C01810=1071.589,307.374,406.167,174.565,30.421,155.473
C01811=1071.583,307.126,406.199,174.562,30.417,155.473
C01812=1071.577,306.878,406.231,174.558,30.412,155.472
C01813=1071.571,306.630,406.263,174.556,30.408,155.471
C01814=1071.564,306.382,406.295,174.552,30.403,155.470
C01815=1071.559,306.135,406.327,174.550,30.399,155.470
C01816=1071.553,305.887,406.359,174.547,30.395,155.469
C01817=1071.547,305.638,406.391,174.543,30.390,155.468
C01818=1071.540,305.390,406.422,174.541,30.386,155.467
C01819=1071.535,305.143,406.454,174.538,30.382,155.467
C01820=1071.529,304.895,406.487,174.535,30.377,155.466
C01821=1071.523,304.647,406.519,174.532,30.373,155.465
C01822=1071.516,304.400,406.550,174.529,30.368,155.464
C01823=1071.510,304.152,406.582,174.526,30.364,155.463
C01824=1071.503,303.847,406.621,174.522,30.359,155.463
C01825=1071.496,303.543,406.660,174.519,30.354,155.462
C01826=1071.488,303.240,406.699,174.515,30.348,155.461
C01827=1071.481,302.936,406.737,174.512,30.343,155.460
C01828=1071.475,302.687,406.769,174.508,30.338,155.459
C01829=1071.469,302.439,406.801,174.506,30.334,155.458
C01830=1071.463,302.192,406.833,174.503,30.330,155.457
C01831=1071.457,301.944,406.865,174.499,30.325,155.457
C01832=1071.452,301.696,406.896,174.497,30.321,155.456
C01833=1071.445,301.448,406.928,174.494,30.317,155.455
C01834=1071.440,301.201,406.959,174.492,30.313,155.454
C01835=1071.434,300.952,406.991,174.488,30.308,155.454
C01836=1071.427,300.704,407.022,174.485,30.304,155.453
C01837=1071.422,300.457,407.054,174.483,30.299,155.452
C01838=1071.416,300.208,407.086,174.479,30.295,155.451
C01839=1071.410,299.961,407.117,174.477,30.291,155.451
C01840=1071.404,299.713,407.149,174.474,30.287,155.450
C01841=1071.399,299.465,407.180,174.470,30.282,155.449
C01842=1071.392,299.217,407.211,174.468,30.278,155.448
C01843=1071.387,298.969,407.243,174.465,30.273,155.448
C01844=1071.380,298.721,407.274,174.463,30.270,155.447
C01845=1071.375,298.473,407.305,174.459,30.265,155.446
C01846=1071.369,298.225,407.337,174.456,30.261,155.445
C01847=1071.363,297.978,407.368,174.454,30.256,155.445
C01848=1071.357,297.729,407.400,174.450,30.252,155.444
C01849=1071.352,297.482,407.431,174.448,30.248,155.443
C01850=1071.345,297.234,407.463,174.445,30.243,155.442
C01851=1071.339,296.986,407.493,174.442,30.239,155.442
C01852=1071.333,296.738,407.525,174.439,30.235,155.441
C01853=1071.327,296.490,407.556,174.436,30.231,155.440
C01854=1071.321,296.242,407.588,174.434,30.226,155.439
C01855=1071.316,295.994,407.618,174.431,30.222,155.439
C01856=1071.309,295.746,407.649,174.427,30.218,155.438
C01857=1071.304,295.498,407.681,174.425,30.214,155.437
C01858=1071.297,295.250,407.712,174.422,30.210,155.436
C01859=1071.291,295.002,407.742,174.420,30.205,155.436
C01860=1071.285,294.754,407.773,174.416,30.201,155.435
C01861=1071.279,294.506,407.804,174.414,30.197,155.434
C01862=1071.273,294.259,407.835,174.411,30.193,155.434
C01863=1071.267,294.010,407.866,174.408,30.189,155.433
C01864=1071.262,293.763,407.898,174.405,30.184,155.432
C01865=1071.255,293.514,407.929,174.402,30.180,155.431
C01866=1071.249,293.266,407.959,174.400,30.176,155.431
C01867=1071.243,293.019,407.990,174.397,30.172,155.430
C01868=1071.237,292.771,408.021,174.393,30.167,155.429
C01869=1071.231,292.522,408.052,174.391,30.164,155.429
C01870=1071.225,292.275,408.083,174.388,30.159,155.428
C01871=1071.219,292.027,408.113,174.386,30.155,155.427
C01872=1071.213,291.778,408.144,174.382,30.151,155.426
C01873=1071.208,291.530,408.175,174.379,30.147,155.426
C01874=1071.202,291.283,408.206,174.377,30.143,155.425
C01875=1071.195,291.034,408.237,174.374,30.139,155.424
C01876=1071.190,290.820,408.264,174.372,30.135,155.424
C01877=1071.185,290.605,408.291,174.369,30.131,155.423
C01878=1071.180,290.390,408.316,174.366,30.128,155.422
C01879=1071.174,290.175,408.343,174.365,30.124,155.422
C01880=1071.169,289.960,408.370,174.362,30.120,155.421
C01881=1071.164,289.745,408.397,174.359,30.117,155.420
C01882=1071.159,289.530,408.423,174.357,30.113,155.420
C01883=1071.154,289.315,408.449,174.355,30.109,155.419
C01884=1071.148,289.068,408.480,174.352,30.105,155.419
C01885=1071.142,288.819,408.511,174.349,30.101,155.418
C01886=1071.136,288.571,408.541,174.346,30.097,155.417
C01887=1071.129,288.323,408.572,174.344,30.093,155.416
C01888=1071.124,288.076,408.603,174.341,30.089,155.416
C01889=1071.118,287.828,408.633,174.338,30.085,155.415
C01890=1071.111,287.579,408.664,174.335,30.080,155.414
C01891=1071.106,287.331,408.694,174.332,30.077,155.414
C01892=1071.099,287.084,408.724,174.330,30.073,155.413
C01893=1071.093,286.835,408.755,174.327,30.068,155.412
C01894=1071.087,286.587,408.784,174.324,30.064,155.411
C01895=1071.081,286.339,408.815,174.321,30.060,155.411
C01896=1071.075,286.091,408.845,174.318,30.056,155.410
C01897=1071.069,285.843,408.876,174.316,30.052,155.409
C01898=1071.063,285.595,408.906,174.313,30.048,155.409
C01899=1071.057,285.347,408.936,174.311,30.044,155.408
C01900=1071.052,285.099,408.967,174.307,30.040,155.407
C01901=1071.045,284.851,408.997,174.305,30.035,155.407
C01902=1071.039,284.603,409.028,174.302,30.032,155.406
C01903=1071.034,284.354,409.057,174.299,30.027,155.405
C01904=1071.028,284.107,409.088,174.297,30.023,155.404
C01905=1071.022,283.858,409.118,174.294,30.019,155.404
C01906=1071.015,283.611,409.148,174.291,30.015,155.403
C01907=1071.009,283.363,409.179,174.288,30.011,155.402
C01908=1071.004,283.114,409.208,174.286,30.007,155.402
C01909=1070.998,282.867,409.239,174.283,30.003,155.401
C01910=1070.991,282.618,409.269,174.280,29.999,155.400
C01911=1070.986,282.370,409.299,174.278,29.994,155.399
C01912=1070.980,282.122,409.329,174.275,29.991,155.399
C01913=1070.974,281.874,409.360,174.272,29.986,155.398
C01914=1070.969,281.625,409.389,174.269,29.982,155.397
C01915=1070.962,281.378,409.419,174.266,29.978,155.397
C01916=1070.956,281.129,409.450,174.264,29.974,155.396
C01917=1070.950,280.881,409.479,174.261,29.970,155.395
C01918=1070.945,280.633,409.510,174.259,29.966,155.395
C01919=1070.939,280.385,409.540,174.256,29.962,155.394
C01920=1070.932,280.137,409.569,174.254,29.958,155.393
C01921=1070.927,279.889,409.599,174.251,29.954,155.393
C01922=1070.921,279.641,409.629,174.248,29.949,155.392
C01923=1070.914,279.393,409.659,174.245,29.945,155.391
C01924=1070.908,279.144,409.689,174.242,29.942,155.391
C01925=1070.903,278.896,409.719,174.240,29.937,155.390
C01926=1070.896,278.648,409.748,174.237,29.933,155.389
C01927=1070.891,278.401,409.779,174.235,29.929,155.388
C01928=1070.885,278.152,409.808,174.232,29.926,155.388
C01929=1070.879,277.904,409.837,174.229,29.921,155.387
C01930=1070.873,277.656,409.868,174.227,29.917,155.386
C01931=1070.867,277.408,409.897,174.223,29.913,155.386
C01932=1070.857,276.988,409.948,174.219,29.906,155.384
C01933=1070.846,276.569,409.998,174.215,29.899,155.383
C01934=1070.836,276.149,410.048,174.210,29.893,155.382
C01935=1070.826,275.729,410.098,174.206,29.886,155.381
C01936=1070.821,275.481,410.128,174.204,29.882,155.380
C01937=1070.814,275.233,410.157,174.200,29.878,155.380
C01938=1070.809,274.985,410.187,174.198,29.873,155.379
C01939=1070.803,274.737,410.216,174.195,29.869,155.378
C01940=1070.797,274.489,410.246,174.192,29.866,155.378
C01941=1070.790,274.241,410.275,174.190,29.862,155.377
C01942=1070.785,273.992,410.305,174.187,29.857,155.376
C01943=1070.779,273.744,410.334,174.185,29.853,155.376
C01944=1070.773,273.496,410.364,174.182,29.849,155.375
C01945=1070.768,273.247,410.393,174.180,29.846,155.374
C01946=1070.761,273.000,410.423,174.177,29.841,155.373
C01947=1070.755,272.752,410.452,174.174,29.837,155.373
C01948=1070.749,272.503,410.482,174.172,29.833,155.372
C01949=1070.743,272.255,410.511,174.169,29.829,155.371
C01950=1070.738,272.007,410.541,174.167,29.826,155.371
C01951=1070.731,271.758,410.570,174.164,29.821,155.370
C01952=1070.725,271.510,410.599,174.162,29.817,155.369
C01953=1070.720,271.262,410.628,174.159,29.813,155.369
C01954=1070.713,271.014,410.657,174.156,29.809,155.368
C01955=1070.708,270.765,410.687,174.153,29.805,155.367
C01956=1070.702,270.517,410.716,174.150,29.801,155.367
C01957=1070.696,270.270,410.745,174.148,29.797,155.366
C01958=1070.690,270.021,410.774,174.145,29.793,155.365
C01959=1070.684,269.773,410.803,174.143,29.789,155.365
C01960=1070.678,269.525,410.832,174.140,29.785,155.364
C01961=1070.672,269.277,410.862,174.138,29.781,155.363
C01962=1070.666,269.028,410.891,174.135,29.777,155.363
C01963=1070.660,268.780,410.920,174.132,29.773,155.362
C01964=1070.654,268.532,410.950,174.130,29.769,155.361
C01965=1070.648,268.284,410.979,174.127,29.765,155.361
C01966=1070.642,268.035,411.007,174.125,29.761,155.360
C01967=1070.636,267.787,411.036,174.122,29.757,155.359
C01968=1070.630,267.539,411.065,174.120,29.753,155.359
C01969=1070.625,267.291,411.094,174.117,29.749,155.358
C01970=1070.619,267.043,411.123,174.115,29.745,155.357
C01971=1070.613,266.794,411.152,174.112,29.741,155.357
C01972=1070.606,266.546,411.181,174.109,29.738,155.356
C01973=1070.601,266.297,411.210,174.107,29.733,155.355
C01974=1070.595,266.049,411.239,174.104,29.729,155.355
C01975=1070.589,265.801,411.268,174.102,29.725,155.354
C01976=1070.583,265.553,411.296,174.099,29.721,155.353
C01977=1070.577,265.305,411.326,174.097,29.717,155.353
C01978=1070.571,265.057,411.355,174.094,29.713,155.352
C01979=1070.565,264.808,411.383,174.092,29.709,155.351
C01980=1070.559,264.560,411.413,174.089,29.705,155.351
C01981=1070.553,264.312,411.442,174.087,29.701,155.350
C01982=1070.547,264.064,411.470,174.084,29.697,155.349
C01983=1070.541,263.815,411.499,174.081,29.694,155.349
C01984=1070.531,263.399,411.547,174.077,29.686,155.347
C01985=1070.521,262.982,411.594,174.073,29.680,155.346
C01986=1070.511,262.566,411.643,174.069,29.673,155.345
C01987=1070.501,262.150,411.691,174.064,29.667,155.344
C01988=1070.495,261.901,411.719,174.062,29.663,155.343
C01989=1070.489,261.654,411.748,174.059,29.659,155.343
C01990=1070.483,261.405,411.776,174.057,29.655,155.342
C01991=1070.477,261.157,411.805,174.054,29.651,155.342
C01992=1070.470,260.909,411.833,174.052,29.647,155.341
C01993=1070.464,260.661,411.862,174.049,29.643,155.340
C01994=1070.458,260.412,411.890,174.047,29.640,155.340
C01995=1070.453,260.164,411.918,174.044,29.636,155.339
C01996=1070.446,259.916,411.947,174.042,29.632,155.338
C01997=1070.440,259.667,411.975,174.040,29.628,155.338
C01998=1070.434,259.419,412.004,174.037,29.624,155.337
C01999=1070.428,259.171,412.032,174.035,29.620,155.336
C02000=1070.422,258.922,412.060,174.032,29.616,155.336
C02001=1070.416,258.674,412.089,174.030,29.612,155.335
C02002=1070.410,258.425,412.117,174.027,29.608,155.334
C02003=1070.405,258.177,412.145,174.025,29.604,155.334
C02004=1070.399,257.929,412.174,174.022,29.601,155.333
C02005=1070.392,257.681,412.202,174.019,29.597,155.332
C02006=1070.386,257.433,412.230,174.017,29.592,155.332
C02007=1070.380,257.184,412.259,174.014,29.588,155.331
C02008=1070.374,256.935,412.287,174.012,29.584,155.330
C02009=1070.369,256.688,412.316,174.009,29.580,155.330
C02010=1070.362,256.439,412.343,174.007,29.576,155.329
C02011=1070.356,256.191,412.372,174.004,29.573,155.328
C02012=1070.351,255.943,412.400,174.003,29.569,155.328
C02013=1070.345,255.694,412.428,174.000,29.565,155.327
C02014=1070.339,255.445,412.456,173.998,29.561,155.326
C02015=1070.333,255.198,412.484,173.995,29.557,155.326
C02016=1070.327,254.949,412.513,173.993,29.553,155.325
C02017=1070.321,254.700,412.541,173.990,29.549,155.325
C02018=1070.315,254.452,412.569,173.988,29.545,155.324
C02019=1070.309,254.204,412.597,173.985,29.541,155.323
C02020=1070.303,253.956,412.625,173.982,29.537,155.322
C02021=1070.297,253.707,412.653,173.980,29.533,155.322
C02022=1070.291,253.458,412.681,173.978,29.529,155.321
C02023=1070.285,253.211,412.709,173.976,29.525,155.320
C02024=1070.279,252.962,412.737,173.973,29.521,155.320
C02025=1070.274,252.714,412.765,173.971,29.517,155.319
C02026=1070.268,252.465,412.793,173.968,29.513,155.318
C02027=1070.261,252.217,412.821,173.966,29.509,155.318
C02028=1070.256,251.969,412.849,173.963,29.505,155.317
C02029=1070.250,251.720,412.877,173.961,29.501,155.316
C02030=1070.245,251.472,412.905,173.958,29.497,155.316
C02031=1070.238,251.223,412.933,173.957,29.494,155.315
C02032=1070.233,250.975,412.961,173.954,29.490,155.315
C02033=1070.227,250.726,412.989,173.952,29.485,155.314
C02034=1070.221,250.478,413.017,173.949,29.481,155.313
C02035=1070.215,250.229,413.044,173.947,29.477,155.312
C02036=1070.205,249.811,413.091,173.942,29.471,155.311
C02037=1070.196,249.392,413.138,173.938,29.464,155.310
C02038=1070.186,248.974,413.185,173.935,29.457,155.309
C02039=1070.176,248.555,413.232,173.931,29.451,155.308
C02040=1070.170,248.307,413.260,173.928,29.446,155.307
C02041=1070.165,248.059,413.288,173.926,29.442,155.307
C02042=1070.159,247.810,413.315,173.923,29.438,155.306
C02043=1070.153,247.562,413.343,173.921,29.434,155.305
C02044=1070.147,247.313,413.371,173.919,29.431,155.305
C02045=1070.142,247.065,413.398,173.917,29.426,155.304
C02046=1070.135,246.816,413.426,173.914,29.422,155.303
C02047=1070.130,246.568,413.454,173.912,29.418,155.303
C02048=1070.124,246.320,413.481,173.909,29.414,155.302
C02049=1070.118,246.071,413.509,173.907,29.410,155.301
C02050=1070.112,245.823,413.536,173.905,29.407,155.301
C02051=1070.107,245.574,413.564,173.902,29.403,155.300
C02052=1070.101,245.326,413.591,173.900,29.399,155.299
C02053=1070.094,245.078,413.619,173.897,29.395,155.299
C02054=1070.089,244.829,413.646,173.895,29.390,155.298
C02055=1070.083,244.581,413.674,173.892,29.386,155.297
C02056=1070.077,244.332,413.701,173.891,29.383,155.297
C02057=1070.071,244.084,413.729,173.888,29.379,155.296
C02058=1070.065,243.835,413.756,173.886,29.375,155.295
C02059=1070.059,243.587,413.784,173.883,29.371,155.295
C02060=1070.054,243.339,413.811,173.881,29.367,155.294
C02061=1070.048,243.090,413.839,173.879,29.363,155.293
C02062=1070.042,242.842,413.865,173.877,29.359,155.293
C02063=1070.037,242.594,413.893,173.874,29.355,155.292
C02064=1070.030,242.345,413.920,173.872,29.351,155.291
C02065=1070.024,242.097,413.948,173.869,29.347,155.291
C02066=1070.018,241.847,413.975,173.868,29.343,155.290
C02067=1070.013,241.599,414.002,173.865,29.339,155.289
C02068=1070.006,241.351,414.030,173.863,29.335,155.289
C02069=1070.000,241.102,414.056,173.860,29.331,155.288
C02070=1069.994,240.854,414.083,173.858,29.327,155.287
C02071=1069.989,240.605,414.111,173.856,29.324,155.287
C02072=1069.983,240.357,414.138,173.854,29.320,155.286
C02073=1069.977,240.108,414.164,173.851,29.316,155.285
C02074=1069.970,239.860,414.192,173.849,29.312,155.285
C02075=1069.965,239.611,414.219,173.846,29.308,155.284
C02076=1069.959,239.363,414.246,173.845,29.304,155.284
C02077=1069.953,239.115,414.274,173.842,29.300,155.283
C02078=1069.947,238.866,414.300,173.840,29.296,155.282
C02079=1069.941,238.618,414.327,173.837,29.292,155.281
C02080=1069.935,238.369,414.354,173.835,29.288,155.281
C02081=1069.930,238.120,414.381,173.833,29.284,155.280
C02082=1069.924,237.872,414.409,173.831,29.280,155.280
C02083=1069.917,237.623,414.436,173.828,29.276,155.279
C02084=1069.912,237.375,414.462,173.826,29.272,155.278
C02085=1069.906,237.127,414.489,173.824,29.268,155.278
C02086=1069.900,236.878,414.516,173.822,29.264,155.277
C02087=1069.894,236.629,414.543,173.819,29.260,155.276
C02088=1069.889,236.417,414.566,173.818,29.257,155.276
C02089=1069.884,236.205,414.589,173.815,29.253,155.275
C02090=1069.879,235.992,414.612,173.813,29.250,155.275
C02091=1069.875,235.780,414.635,173.812,29.247,155.274
C02092=1069.869,235.567,414.658,173.809,29.243,155.273
C02093=1069.864,235.354,414.681,173.808,29.240,155.273
C02094=1069.859,235.142,414.704,173.806,29.236,155.272
C02095=1069.854,234.929,414.727,173.804,29.233,155.272
C02096=1069.848,234.681,414.754,173.801,29.229,155.271
C02097=1069.842,234.432,414.781,173.800,29.225,155.270
C02098=1069.836,234.184,414.808,173.797,29.221,155.270
C02099=1069.830,233.936,414.834,173.795,29.217,155.269
C02100=1069.824,233.687,414.861,173.792,29.213,155.268
C02101=1069.819,233.439,414.888,173.791,29.209,155.268
C02102=1069.813,233.189,414.914,173.788,29.205,155.267
C02103=1069.807,232.941,414.940,173.786,29.201,155.266
C02104=1069.801,232.693,414.967,173.783,29.197,155.266
C02105=1069.795,232.444,414.994,173.782,29.193,155.265
C02106=1069.790,232.196,415.020,173.779,29.189,155.265
C02107=1069.783,231.947,415.047,173.777,29.185,155.264
C02108=1069.777,231.698,415.074,173.775,29.181,155.263
C02109=1069.772,231.450,415.101,173.773,29.177,155.262
C02110=1069.766,231.202,415.127,173.770,29.173,155.262
C02111=1069.760,230.953,415.154,173.768,29.169,155.261
C02112=1069.755,230.704,415.180,173.766,29.166,155.260
C02113=1069.749,230.456,415.207,173.764,29.162,155.260
C02114=1069.743,230.208,415.233,173.761,29.158,155.259
C02115=1069.737,229.959,415.260,173.760,29.154,155.259
C02116=1069.730,229.711,415.286,173.757,29.149,155.258
C02117=1069.725,229.462,415.312,173.755,29.145,155.257
C02118=1069.719,229.213,415.339,173.752,29.141,155.257
C02119=1069.713,228.965,415.366,173.751,29.138,155.256
C02120=1069.707,228.717,415.392,173.748,29.134,155.255
C02121=1069.701,228.467,415.418,173.746,29.130,155.255
C02122=1069.695,228.219,415.445,173.744,29.126,155.254
C02123=1069.689,227.970,415.471,173.742,29.122,155.253
C02124=1069.683,227.722,415.497,173.739,29.118,155.253
C02125=1069.677,227.473,415.523,173.737,29.114,155.252
C02126=1069.671,227.225,415.550,173.735,29.110,155.251
C02127=1069.666,226.976,415.576,173.733,29.106,155.251
C02128=1069.659,226.728,415.602,173.730,29.102,155.250
C02129=1069.654,226.480,415.628,173.729,29.098,155.249
C02130=1069.647,226.230,415.655,173.726,29.094,155.249
C02131=1069.642,225.982,415.681,173.724,29.090,155.248
C02132=1069.635,225.733,415.707,173.722,29.086,155.247
C02133=1069.630,225.485,415.733,173.720,29.082,155.247
C02134=1069.624,225.236,415.759,173.718,29.078,155.246
C02135=1069.618,224.988,415.785,173.716,29.074,155.245
C02136=1069.612,224.739,415.811,173.714,29.070,155.245
C02137=1069.606,224.490,415.838,173.711,29.066,155.244
C02138=1069.600,224.242,415.864,173.710,29.062,155.243
C02139=1069.595,223.993,415.890,173.707,29.058,155.243
C02140=1069.589,223.744,415.916,173.705,29.054,155.242
C02141=1069.583,223.496,415.942,173.703,29.050,155.241
C02142=1069.577,223.247,415.968,173.701,29.046,155.241
C02143=1069.571,222.999,415.995,173.698,29.042,155.240
C02144=1069.566,222.783,416.017,173.697,29.039,155.239
C02145=1069.561,222.566,416.040,173.695,29.035,155.239
C02146=1069.556,222.350,416.062,173.693,29.031,155.238
C02147=1069.551,222.132,416.085,173.691,29.028,155.238
C02148=1069.546,221.916,416.107,173.690,29.025,155.237
C02149=1069.541,221.699,416.131,173.687,29.021,155.237
C02150=1069.536,221.483,416.153,173.686,29.018,155.236
C02151=1069.531,221.266,416.176,173.684,29.015,155.235
C02152=1069.525,221.017,416.201,173.682,29.010,155.235
C02153=1069.519,220.768,416.227,173.679,29.006,155.234
C02154=1069.513,220.520,416.253,173.678,29.002,155.233
C02155=1069.507,220.271,416.279,173.675,28.998,155.233
C02156=1069.501,220.023,416.304,173.673,28.994,155.232
C02157=1069.494,219.775,416.331,173.671,28.991,155.231
C02158=1069.489,219.526,416.356,173.669,28.987,155.231
C02159=1069.483,219.277,416.382,173.667,28.983,155.230
C02160=1069.477,219.028,416.408,173.665,28.979,155.230
C02161=1069.471,218.780,416.434,173.662,28.975,155.229
C02162=1069.465,218.531,416.460,173.661,28.970,155.228
C02163=1069.459,218.282,416.485,173.658,28.966,155.227
C02164=1069.453,218.034,416.510,173.656,28.962,155.227
C02165=1069.448,217.785,416.536,173.654,28.959,155.226
C02166=1069.441,217.537,416.562,173.652,28.955,155.226
C02167=1069.436,217.288,416.588,173.650,28.951,155.225
C02168=1069.430,217.040,416.613,173.648,28.947,155.224
C02169=1069.424,216.791,416.639,173.646,28.942,155.223
C02170=1069.418,216.542,416.665,173.644,28.939,155.223
C02171=1069.412,216.293,416.690,173.642,28.935,155.222
C02172=1069.406,216.044,416.716,173.639,28.931,155.222
C02173=1069.401,215.796,416.741,173.638,28.927,155.221
C02174=1069.395,215.548,416.766,173.635,28.922,155.220
C02175=1069.389,215.299,416.793,173.634,28.919,155.219
C02176=1069.383,215.051,416.818,173.631,28.914,155.219
C02177=1069.377,214.802,416.844,173.629,28.910,155.218
C02178=1069.371,214.553,416.869,173.627,28.907,155.218
C02179=1069.365,214.305,416.894,173.625,28.902,155.217
C02180=1069.360,214.056,416.920,173.624,28.898,155.216
C02181=1069.354,213.808,416.946,173.621,28.894,155.215
C02182=1069.348,213.559,416.971,173.619,28.890,155.215
C02183=1069.342,213.310,416.997,173.617,28.886,155.214
C02184=1069.336,213.062,417.022,173.615,28.882,155.213
C02185=1069.330,212.813,417.047,173.613,28.878,155.213
C02186=1069.325,212.564,417.073,173.611,28.874,155.212
C02187=1069.319,212.315,417.098,173.608,28.870,155.211
C02188=1069.313,212.066,417.123,173.607,28.866,155.211
C02189=1069.306,211.818,417.148,173.605,28.862,155.210
C02190=1069.301,211.570,417.173,173.603,28.858,155.209
C02191=1069.295,211.321,417.199,173.601,28.854,155.209
C02192=1069.289,211.072,417.225,173.599,28.850,155.208
C02193=1069.283,210.823,417.250,173.597,28.846,155.207
C02194=1069.277,210.575,417.275,173.594,28.842,155.207
C02195=1069.271,210.326,417.300,173.593,28.838,155.206
C02196=1069.265,210.077,417.325,173.590,28.834,155.205
C02197=1069.260,209.828,417.351,173.589,28.830,155.205
C02198=1069.254,209.580,417.376,173.587,28.826,155.204
C02199=1069.248,209.332,417.401,173.585,28.822,155.203
C02200=1069.243,209.117,417.423,173.583,28.818,155.203
C02201=1069.237,208.903,417.444,173.581,28.815,155.202
C02202=1069.232,208.688,417.466,173.580,28.811,155.202
C02203=1069.228,208.474,417.487,173.578,28.808,155.201
C02204=1069.223,208.259,417.509,173.576,28.804,155.200
C02205=1069.218,208.046,417.531,173.574,28.801,155.200
C02206=1069.212,207.831,417.552,173.572,28.798,155.199
C02207=1069.207,207.616,417.574,173.571,28.794,155.199
C02208=1069.183,206.573,417.677,173.428,28.722,155.196
C02209=1069.177,206.324,417.701,173.427,28.718,155.195
C02210=1069.171,206.076,417.725,173.424,28.715,155.195
C02211=1069.166,205.827,417.749,173.422,28.712,155.194
C02212=1069.160,205.578,417.774,173.420,28.709,155.194
C02213=1069.155,205.329,417.798,173.418,28.706,155.193
C02214=1069.148,205.080,417.822,173.415,28.703,155.193
C02215=1069.143,204.832,417.846,173.414,28.700,155.192
C02216=1069.138,204.583,417.871,173.411,28.697,155.192
C02217=1069.132,204.334,417.895,173.409,28.693,155.191
C02218=1069.126,204.086,417.919,173.407,28.690,155.191
C02219=1069.120,203.837,417.943,173.404,28.687,155.190
C02220=1069.115,203.588,417.968,173.402,28.684,155.190
C02221=1069.109,203.339,417.992,173.400,28.681,155.190
C02222=1069.103,203.091,418.016,173.398,28.678,155.189
C02223=1069.097,202.842,418.040,173.395,28.675,155.189
C02224=1069.092,202.593,418.065,173.394,28.672,155.188
C02225=1069.087,202.344,418.089,173.391,28.669,155.188
C02226=1069.080,202.095,418.113,173.389,28.665,155.187
C02227=1069.075,201.847,418.137,173.387,28.662,155.187
C02228=1069.069,201.598,418.160,173.384,28.660,155.187
C02229=1069.063,201.349,418.185,173.382,28.656,155.186
C02230=1069.057,201.100,418.208,173.380,28.653,155.186
C02231=1069.052,200.852,418.233,173.378,28.650,155.185
C02232=1069.045,200.603,418.257,173.376,28.647,155.185
C02233=1069.040,200.354,418.281,173.374,28.644,155.184
C02234=1069.034,200.105,418.304,173.371,28.641,155.184
C02235=1069.028,199.856,418.328,173.370,28.638,155.183
C02236=1069.022,199.608,418.352,173.367,28.635,155.183
C02237=1069.017,199.359,418.376,173.364,28.632,155.183
C02238=1069.011,199.110,418.400,173.363,28.629,155.182
C02239=1069.005,198.861,418.423,173.360,28.626,155.182
C02240=1068.999,198.613,418.448,173.359,28.623,155.181
C02241=1068.993,198.364,418.472,173.356,28.620,155.181
C02242=1068.988,198.115,418.495,173.354,28.617,155.180
C02243=1068.982,197.866,418.519,173.352,28.614,155.180
C02244=1068.976,197.618,418.543,173.350,28.611,155.180
C02245=1068.970,197.368,418.566,173.348,28.608,155.179
C02246=1068.965,197.119,418.591,173.345,28.605,155.179
C02247=1068.959,196.871,418.614,173.343,28.602,155.178
C02248=1068.952,196.622,418.638,173.341,28.599,155.178
C02249=1068.947,196.373,418.662,173.339,28.596,155.177
C02250=1068.941,196.125,418.685,173.337,28.593,155.177
C02251=1068.936,195.876,418.709,173.335,28.590,155.177
C02252=1068.930,195.627,418.733,173.332,28.587,155.176
C02253=1068.924,195.378,418.757,173.331,28.584,155.176
C02254=1068.918,195.129,418.780,173.328,28.581,155.175
C02255=1068.912,194.881,418.804,173.326,28.578,155.175
C02256=1068.907,194.632,418.827,173.324,28.575,155.174
C02257=1068.901,194.383,418.851,173.322,28.572,155.174
C02258=1068.896,194.133,418.875,173.320,28.569,155.173
C02259=1068.890,193.885,418.899,173.317,28.566,155.173
C02260=1068.884,193.636,418.922,173.316,28.563,155.173
C02261=1068.879,193.388,418.946,173.313,28.560,155.172
C02262=1068.873,193.139,418.969,173.312,28.557,155.172
C02263=1068.868,192.890,418.993,173.309,28.554,155.171
C02264=1068.861,192.641,419.016,173.307,28.551,155.171
C02265=1068.855,192.392,419.040,173.305,28.548,155.170
C02266=1068.850,192.143,419.064,173.303,28.545,155.170
C02267=1068.844,191.895,419.087,173.301,28.542,155.170
C02268=1068.838,191.646,419.110,173.298,28.538,155.169
C02269=1068.832,191.363,419.138,173.297,28.536,155.169
C02270=1068.826,191.081,419.164,173.294,28.532,155.168
C02271=1068.819,190.799,419.191,173.292,28.529,155.168
C02272=1068.813,190.517,419.217,173.289,28.525,155.167
C02273=1068.808,190.268,419.241,173.287,28.522,155.167
C02274=1068.802,190.020,419.264,173.285,28.519,155.166
C02275=1068.796,189.771,419.287,173.283,28.516,155.166
C02276=1068.791,189.521,419.311,173.281,28.513,155.165
C02277=1068.785,189.273,419.334,173.279,28.510,155.165
C02278=1068.779,189.024,419.357,173.277,28.507,155.165
C02279=1068.774,188.775,419.381,173.274,28.504,155.164
C02280=1068.768,188.526,419.405,173.273,28.501,155.164
C02281=1068.762,188.277,419.428,173.270,28.498,155.163
C02282=1068.757,188.028,419.451,173.269,28.495,155.163
C02283=1068.751,187.779,419.474,173.266,28.492,155.162
C02284=1068.745,187.531,419.498,173.265,28.489,155.162
C02285=1068.739,187.282,419.521,173.262,28.486,155.161
C02286=1068.734,187.033,419.544,173.261,28.483,155.161
C02287=1068.729,186.784,419.567,173.258,28.480,155.161
C02288=1068.723,186.536,419.591,173.257,28.477,155.160
C02289=1068.718,186.286,419.615,173.254,28.474,155.160
C02290=1068.712,186.037,419.638,173.252,28.471,155.159
C02291=1068.706,185.789,419.661,173.250,28.468,155.159
C02292=1068.700,185.540,419.683,173.248,28.465,155.158
C02293=1068.695,185.291,419.708,173.246,28.462,155.158
C02294=1068.689,185.042,419.731,173.244,28.459,155.158
C02295=1068.684,184.793,419.754,173.242,28.456,155.157
C02296=1068.678,184.544,419.777,173.240,28.453,155.157
C02297=1068.672,184.295,419.800,173.238,28.450,155.156
C02298=1068.666,184.047,419.822,173.236,28.448,155.156
C02299=1068.661,183.798,419.845,173.233,28.445,155.156
C02300=1068.655,183.549,419.868,173.232,28.442,155.155
C02301=1068.649,183.300,419.891,173.229,28.439,155.155
C02302=1068.644,183.051,419.914,173.228,28.436,155.154
C02303=1068.637,182.802,419.937,173.225,28.433,155.154
C02304=1068.631,182.554,419.960,173.224,28.430,155.153
C02305=1068.626,182.305,419.982,173.221,28.427,155.153
C02306=1068.620,182.056,420.005,173.220,28.424,155.153
C02307=1068.614,181.807,420.028,173.218,28.422,155.152
C02308=1068.608,181.558,420.051,173.215,28.419,155.152
C02309=1068.602,181.309,420.074,173.214,28.416,155.151
C02310=1068.596,181.060,420.097,173.211,28.413,155.151
C02311=1068.591,180.812,420.120,173.210,28.410,155.151
C02312=1068.585,180.563,420.143,173.207,28.407,155.150
C02313=1068.579,180.314,420.165,173.206,28.405,155.150
C02314=1068.573,180.065,420.188,173.203,28.402,155.149
C02315=1068.567,179.816,420.211,173.201,28.399,155.149
C02316=1068.561,179.567,420.234,173.199,28.396,155.149
C02317=1068.556,179.318,420.256,173.197,28.393,155.148
C02318=1068.550,179.069,420.279,173.195,28.390,155.148
C02319=1068.544,178.820,420.302,173.193,28.387,155.147
C02320=1068.538,178.571,420.324,173.192,28.385,155.147
C02321=1068.532,178.323,420.347,173.189,28.382,155.147
C02322=1068.526,178.074,420.370,173.187,28.379,155.146
C02323=1068.521,177.825,420.393,173.185,28.376,155.146
C02324=1068.515,177.575,420.415,173.183,28.373,155.145
C02325=1068.509,177.327,420.438,173.181,28.370,155.145
C02326=1068.503,177.078,420.461,173.179,28.367,155.145
C02327=1068.497,176.829,420.483,173.178,28.364,155.144
C02328=1068.492,176.579,420.506,173.175,28.361,155.144
C02329=1068.485,176.331,420.528,173.174,28.359,155.143
C02330=1068.480,176.082,420.551,173.171,28.356,155.143
C02331=1068.474,175.834,420.574,173.169,28.353,155.143
C02332=1068.469,175.584,420.596,173.167,28.350,155.142
C02333=1068.462,175.301,420.621,173.165,28.347,155.142
C02334=1068.456,175.019,420.647,173.163,28.344,155.141
C02335=1068.449,174.736,420.673,173.160,28.340,155.141
C02336=1068.442,174.454,420.698,173.158,28.337,155.140
C02337=1068.437,174.205,420.721,173.156,28.334,155.140
C02338=1068.431,173.956,420.744,173.155,28.331,155.139
C02339=1068.425,173.707,420.766,173.152,28.328,155.139
C02340=1068.420,173.459,420.788,173.151,28.326,155.139
C02341=1068.414,173.210,420.811,173.148,28.323,155.138
C02342=1068.408,172.960,420.833,173.147,28.320,155.138
C02343=1068.402,172.712,420.856,173.145,28.317,155.137
C02344=1068.397,172.462,420.878,173.143,28.314,155.137
C02345=1068.391,172.213,420.901,173.141,28.311,155.137
C02346=1068.385,171.965,420.923,173.139,28.309,155.136
C02347=1068.380,171.716,420.945,173.137,28.306,155.136
C02348=1068.374,171.467,420.968,173.135,28.303,155.135
C02349=1068.368,171.217,420.990,173.133,28.299,155.135
C02350=1068.363,170.970,421.012,173.131,28.297,155.135
C02351=1068.357,170.720,421.034,173.130,28.294,155.134
C02352=1068.351,170.471,421.057,173.127,28.291,155.134
C02353=1068.345,170.222,421.079,173.126,28.288,155.133
C02354=1068.339,169.973,421.102,173.123,28.285,155.133
C02355=1068.335,169.724,421.124,173.121,28.283,155.133
C02356=1068.328,169.476,421.146,173.120,28.280,155.132
C02357=1068.323,169.226,421.168,173.117,28.277,155.132
C02358=1068.318,168.978,421.191,173.116,28.274,155.131
C02359=1068.311,168.729,421.213,173.114,28.271,155.131
C02360=1068.306,168.480,421.236,173.112,28.268,155.130
C02361=1068.300,168.230,421.258,173.110,28.265,155.130
C02362=1068.294,167.982,421.280,173.109,28.262,155.130
C02363=1068.289,167.733,421.302,173.106,28.259,155.129
C02364=1068.284,167.483,421.324,173.104,28.257,155.129
C02365=1068.278,167.235,421.346,173.103,28.254,155.128
C02366=1068.272,166.986,421.368,173.100,28.251,155.128
C02367=1068.267,166.737,421.391,173.099,28.248,155.128
C02368=1068.260,166.488,421.413,173.097,28.245,155.127
C02369=1068.256,166.239,421.435,173.095,28.242,155.127
C02370=1068.250,165.990,421.458,173.093,28.239,155.126
C02371=1068.244,165.742,421.479,173.092,28.236,155.126
C02372=1068.239,165.492,421.501,173.089,28.233,155.125
C02373=1068.233,165.243,421.524,173.088,28.231,155.125
C02374=1068.228,164.995,421.546,173.086,28.228,155.125
C02375=1068.222,164.745,421.568,173.083,28.225,155.124
C02376=1068.216,164.497,421.590,173.082,28.222,155.124
C02377=1068.211,164.248,421.612,173.080,28.219,155.123
C02378=1068.205,163.998,421.634,173.078,28.216,155.123
C02379=1068.199,163.749,421.656,173.076,28.213,155.123
C02380=1068.194,163.501,421.678,173.075,28.211,155.122
C02381=1068.188,163.252,421.700,173.072,28.208,155.122
C02382=1068.183,163.003,421.722,173.071,28.205,155.121
C02383=1068.178,162.753,421.744,173.069,28.202,155.121
C02384=1068.171,162.505,421.767,173.067,28.199,155.120
C02385=1068.166,162.256,421.788,173.065,28.196,155.120
C02386=1068.160,162.007,421.810,173.064,28.193,155.120
C02387=1068.155,161.758,421.832,173.061,28.190,155.119
C02388=1068.150,161.508,421.854,173.059,28.187,155.119
C02389=1068.144,161.260,421.875,173.058,28.185,155.118
C02390=1068.139,161.011,421.898,173.055,28.182,155.118
C02391=1068.133,160.762,421.920,173.054,28.179,155.118
C02392=1068.127,160.513,421.941,173.052,28.176,155.117
C02393=1068.121,160.264,421.963,173.051,28.173,155.117
C02394=1068.115,160.015,421.985,173.048,28.170,155.116
C02395=1068.110,159.766,422.006,173.047,28.168,155.116
C02396=1068.104,159.517,422.028,173.045,28.165,155.116
C02397=1068.097,159.234,422.052,173.043,28.161,155.115
C02398=1068.091,158.950,422.078,173.040,28.158,155.115
C02399=1068.085,158.668,422.102,173.039,28.155,155.114
C02400=1068.078,158.385,422.126,173.036,28.152,155.114
C02401=1068.072,158.136,422.148,173.035,28.149,155.113
C02402=1068.066,157.887,422.170,173.033,28.147,155.113
C02403=1068.061,157.638,422.192,173.030,28.144,155.113
C02404=1068.055,157.389,422.213,173.029,28.141,155.112
C02405=1068.049,157.140,422.234,173.027,28.138,155.112
C02406=1068.043,156.891,422.256,173.026,28.135,155.111
C02407=1068.038,156.642,422.278,173.023,28.132,155.111
C02408=1068.032,156.393,422.300,173.022,28.130,155.111
C02409=1068.026,156.144,422.321,173.020,28.127,155.110
C02410=1068.020,155.895,422.342,173.018,28.124,155.110
C02411=1068.015,155.646,422.365,173.016,28.121,155.109
C02412=1068.009,155.397,422.386,173.014,28.118,155.109
C02413=1068.003,155.148,422.408,173.013,28.116,155.109
C02414=1067.998,154.899,422.429,173.010,28.113,155.108
C02415=1067.992,154.650,422.450,173.009,28.110,155.108
C02416=1067.986,154.402,422.472,173.007,28.107,155.107
C02417=1067.980,154.152,422.493,173.006,28.104,155.107
C02418=1067.974,153.903,422.514,173.003,28.101,155.107
C02419=1067.969,153.654,422.536,173.002,28.099,155.106
C02420=1067.963,153.405,422.558,173.000,28.096,155.106
C02421=1067.957,153.156,422.579,172.998,28.093,155.105
C02422=1067.951,152.907,422.601,172.996,28.090,155.105
C02423=1067.946,152.658,422.621,172.994,28.087,155.105
C02424=1067.940,152.409,422.643,172.993,28.085,155.104
C02425=1067.934,152.160,422.664,172.990,28.082,155.104
C02426=1067.928,151.911,422.686,172.989,28.079,155.104
C02427=1067.923,151.662,422.706,172.987,28.077,155.103
C02428=1067.917,151.413,422.728,172.986,28.074,155.103
C02429=1067.912,151.164,422.750,172.983,28.071,155.102
C02430=1067.906,150.914,422.772,172.982,28.068,155.102
C02431=1067.900,150.665,422.792,172.980,28.065,155.102
C02432=1067.894,150.416,422.814,172.978,28.063,155.101
C02433=1067.889,150.168,422.835,172.976,28.060,155.101
C02434=1067.883,149.919,422.856,172.974,28.057,155.100
C02435=1067.877,149.669,422.877,172.973,28.054,155.100
C02436=1067.872,149.421,422.898,172.971,28.051,155.100
C02437=1067.866,149.172,422.920,172.970,28.049,155.099
C02438=1067.860,148.923,422.941,172.967,28.046,155.099
C02439=1067.854,148.673,422.962,172.966,28.043,155.098
C02440=1067.849,148.424,422.983,172.964,28.040,155.098
C02441=1067.843,148.175,423.004,172.963,28.037,155.098
C02442=1067.837,147.926,423.026,172.960,28.034,155.097
C02443=1067.831,147.677,423.047,172.959,28.032,155.097
C02444=1067.826,147.428,423.068,172.957,28.029,155.096
C02445=1067.820,147.179,423.088,172.955,28.026,155.096
C02446=1067.814,146.930,423.109,172.954,28.023,155.095
C02447=1067.808,146.682,423.131,172.951,28.021,155.095
C02448=1067.802,146.432,423.152,172.950,28.018,155.095
C02449=1067.797,146.183,423.173,172.948,28.015,155.094
C02450=1067.791,145.933,423.194,172.947,28.013,155.094
C02451=1067.785,145.685,423.215,172.944,28.010,155.094
C02452=1067.779,145.435,423.235,172.943,28.007,155.093
C02453=1067.773,145.187,423.257,172.941,28.004,155.093
C02454=1067.768,144.938,423.277,172.939,28.001,155.092
C02455=1067.762,144.689,423.299,172.938,27.999,155.092
C02456=1067.756,144.439,423.319,172.935,27.996,155.092
C02457=1067.750,144.190,423.341,172.934,27.993,155.091
C02458=1067.744,143.941,423.361,172.932,27.991,155.091
C02459=1067.739,143.693,423.382,172.931,27.988,155.091
C02460=1067.733,143.443,423.403,172.929,27.985,155.090
C02461=1067.727,143.160,423.427,172.927,27.982,155.090
C02462=1067.719,142.877,423.451,172.925,27.979,155.089
C02463=1067.713,142.594,423.474,172.923,27.975,155.089
C02464=1067.707,142.310,423.498,172.921,27.973,155.088
C02465=1067.701,142.061,423.520,172.919,27.970,155.088
C02466=1067.696,141.812,423.540,172.917,27.967,155.088
C02467=1067.689,141.563,423.560,172.916,27.964,155.087
C02468=1067.684,141.314,423.582,172.914,27.961,155.087
C02469=1067.678,141.065,423.602,172.913,27.958,155.086
C02470=1067.673,140.815,423.623,172.910,27.955,155.086
C02471=1067.667,140.567,423.644,172.908,27.953,155.086
C02472=1067.661,140.318,423.664,172.907,27.950,155.085
C02473=1067.655,140.068,423.685,172.905,27.947,155.085
C02474=1067.650,139.820,423.707,172.904,27.944,155.084
C02475=1067.644,139.571,423.727,172.902,27.942,155.084
C02476=1067.638,139.321,423.747,172.900,27.939,155.084
C02477=1067.632,139.073,423.769,172.898,27.936,155.083
C02478=1067.626,138.824,423.789,172.897,27.934,155.083
C02479=1067.620,138.574,423.810,172.895,27.931,155.082
C02480=1067.615,138.325,423.830,172.894,27.928,155.082
C02481=1067.609,138.077,423.851,172.892,27.925,155.082
C02482=1067.604,137.828,423.871,172.890,27.922,155.081
C02483=1067.598,137.578,423.892,172.888,27.920,155.081
C02484=1067.592,137.329,423.912,172.886,27.917,155.080
C02485=1067.586,137.080,423.933,172.885,27.914,155.080
C02486=1067.580,136.831,423.954,172.883,27.911,155.080
C02487=1067.574,136.582,423.974,172.882,27.909,155.079
C02488=1067.568,136.333,423.994,172.879,27.906,155.079
C02489=1067.562,136.083,424.015,172.878,27.903,155.079
C02490=1067.557,135.834,424.036,172.876,27.901,155.078
C02491=1067.551,135.585,424.056,172.875,27.898,155.078
C02492=1067.546,135.337,424.077,172.873,27.895,155.077
C02493=1067.539,135.087,424.097,172.872,27.892,155.077
C02494=1067.534,134.838,424.118,172.869,27.889,155.077
C02495=1067.528,134.589,424.138,172.867,27.886,155.076
C02496=1067.522,134.340,424.158,172.866,27.884,155.076
C02497=1067.517,134.090,424.179,172.864,27.881,155.075
C02498=1067.511,133.841,424.199,172.863,27.879,155.075
C02499=1067.505,133.592,424.220,172.861,27.876,155.075
C02500=1067.499,133.344,424.240,172.860,27.873,155.074
C02501=1067.494,133.094,424.260,172.857,27.870,155.074
C02502=1067.487,132.846,424.281,172.856,27.867,155.073
C02503=1067.482,132.596,424.302,172.854,27.865,155.073
C02504=1067.476,132.348,424.322,172.853,27.862,155.073
C02505=1067.471,132.098,424.343,172.851,27.859,155.072
C02506=1067.464,131.849,424.363,172.850,27.856,155.072
C02507=1067.459,131.600,424.383,172.848,27.854,155.071
C02508=1067.453,131.351,424.403,172.846,27.851,155.071
C02509=1067.447,131.102,424.423,172.844,27.848,155.071
C02510=1067.441,130.852,424.444,172.842,27.846,155.070
C02511=1067.435,130.603,424.463,172.841,27.843,155.070
C02512=1067.429,130.354,424.483,172.839,27.840,155.070
C02513=1067.424,130.105,424.504,172.838,27.837,155.069
C02514=1067.418,129.855,424.524,172.836,27.835,155.069
C02515=1067.412,129.607,424.544,172.834,27.832,155.068
C02516=1067.406,129.358,424.564,172.832,27.829,155.068
C02517=1067.400,129.109,424.585,172.831,27.826,155.068
C02518=1067.394,128.860,424.605,172.829,27.824,155.067
C02519=1067.388,128.610,424.625,172.827,27.821,155.067
C02520=1067.382,128.361,424.646,172.826,27.819,155.067
C02521=1067.377,128.112,424.665,172.824,27.816,155.066
C02522=1067.371,127.863,424.685,172.823,27.813,155.066
C02523=1067.365,127.614,424.705,172.820,27.810,155.065
C02524=1067.359,127.364,424.726,172.819,27.807,155.065
C02525=1067.352,127.081,424.749,172.817,27.805,155.065
C02526=1067.345,126.798,424.771,172.816,27.802,155.064
C02527=1067.339,126.515,424.794,172.813,27.798,155.064
C02528=1067.332,126.231,424.816,172.812,27.795,155.063
C02529=1067.326,125.982,424.836,172.810,27.793,155.063
C02530=1067.321,125.733,424.857,172.808,27.790,155.063
C02531=1067.315,125.484,424.877,172.806,27.787,155.062
C02532=1067.309,125.235,424.896,172.805,27.784,155.062
C02533=1067.303,124.985,424.916,172.803,27.781,155.061
C02534=1067.297,124.737,424.936,172.802,27.779,155.061
C02535=1067.291,124.487,424.957,172.800,27.776,155.061
C02536=1067.286,124.238,424.976,172.799,27.774,155.060
C02537=1067.280,123.989,424.996,172.797,27.771,155.060
C02538=1067.274,123.740,425.016,172.795,27.768,155.059
C02539=1067.269,123.491,425.036,172.794,27.765,155.059
C02540=1067.263,123.242,425.056,172.791,27.762,155.059
C02541=1067.257,122.993,425.076,172.790,27.759,155.058
C02542=1067.251,122.744,425.095,172.788,27.757,155.058
C02543=1067.244,122.494,425.115,172.787,27.754,155.058
C02544=1067.239,122.245,425.136,172.785,27.752,155.057
C02545=1067.233,121.995,425.155,172.784,27.749,155.057
C02546=1067.227,121.747,425.175,172.782,27.746,155.056
C02547=1067.221,121.498,425.195,172.781,27.743,155.056
C02548=1067.216,121.248,425.214,172.779,27.741,155.056
C02549=1067.211,120.999,425.235,172.778,27.738,155.055
C02550=1067.205,120.750,425.255,172.776,27.735,155.055
C02551=1067.199,120.501,425.274,172.774,27.732,155.054
C02552=1067.193,120.252,425.294,172.772,27.729,155.054
C02553=1067.187,120.003,425.313,172.771,27.726,155.054
C02554=1067.182,119.754,425.334,172.769,27.724,155.053
C02555=1067.176,119.504,425.353,172.768,27.721,155.053
C02556=1067.170,119.255,425.373,172.766,27.719,155.052
C02557=1067.164,119.007,425.393,172.764,27.716,155.052
C02558=1067.159,118.757,425.412,172.763,27.713,155.052
C02559=1067.153,118.508,425.432,172.761,27.710,155.051
C02560=1067.148,118.259,425.452,172.760,27.708,155.051
C02561=1067.142,118.010,425.472,172.758,27.705,155.050
C02562=1067.136,117.760,425.491,172.757,27.702,155.050
C02563=1067.130,117.512,425.511,172.755,27.699,155.050
C02564=1067.124,117.262,425.531,172.754,27.696,155.049
C02565=1067.118,117.013,425.551,172.751,27.693,155.049
C02566=1067.113,116.764,425.570,172.750,27.691,155.048
C02567=1067.107,116.515,425.590,172.748,27.688,155.048
C02568=1067.102,116.265,425.610,172.747,27.685,155.048
C02569=1067.096,116.016,425.629,172.745,27.682,155.047
C02570=1067.090,115.767,425.649,172.744,27.679,155.047
C02571=1067.084,115.518,425.668,172.742,27.677,155.046
C02572=1067.078,115.269,425.688,172.741,27.674,155.046
C02573=1067.073,115.019,425.707,172.739,27.671,155.046
C02574=1067.067,114.770,425.728,172.738,27.668,155.045
C02575=1067.062,114.522,425.747,172.736,27.666,155.045
C02576=1067.057,114.272,425.766,172.735,27.663,155.044
C02577=1067.051,114.023,425.786,172.733,27.660,155.044
C02578=1067.045,113.774,425.805,172.731,27.657,155.044
C02579=1067.039,113.524,425.824,172.730,27.655,155.043
C02580=1067.033,113.276,425.844,172.728,27.652,155.043
C02581=1067.027,113.027,425.863,172.727,27.649,155.042
C02582=1067.021,112.777,425.882,172.724,27.646,155.042
C02583=1067.015,112.528,425.902,172.723,27.644,155.042
C02584=1067.009,112.279,425.921,172.721,27.641,155.041
C02585=1067.004,112.029,425.941,172.720,27.638,155.041
C02586=1066.998,111.781,425.961,172.718,27.635,155.041
C02587=1066.992,111.531,425.980,172.717,27.632,155.040
C02588=1066.986,111.282,425.999,172.715,27.630,155.040
C02589=1066.979,110.998,426.021,172.714,27.627,155.039
C02590=1066.973,110.715,426.043,172.712,27.624,155.039
C02591=1066.967,110.432,426.065,172.710,27.620,155.038
C02592=1066.959,110.148,426.087,172.708,27.618,155.038
C02593=1066.954,109.899,426.106,172.707,27.615,155.038
C02594=1066.948,109.650,426.125,172.705,27.612,155.037
C02595=1066.941,109.400,426.144,172.704,27.610,155.037
C02596=1066.936,109.151,426.163,172.702,27.607,155.037
C02597=1066.930,108.902,426.183,172.701,27.604,155.036
C02598=1066.924,108.653,426.202,172.699,27.601,155.036
C02599=1066.919,108.404,426.221,172.698,27.599,155.035
C02600=1066.913,108.155,426.240,172.696,27.596,155.035
C02601=1066.907,107.905,426.259,172.695,27.593,155.035
C02602=1066.901,107.656,426.278,172.692,27.591,155.034
C02603=1066.895,107.407,426.298,172.691,27.588,155.034
C02604=1066.889,107.158,426.317,172.689,27.585,155.033
C02605=1066.883,106.909,426.336,172.688,27.582,155.033
C02606=1066.877,106.659,426.356,172.686,27.579,155.033
C02607=1066.871,106.410,426.374,172.685,27.577,155.032
C02608=1066.866,106.161,426.393,172.683,27.574,155.032
C02609=1066.860,105.912,426.412,172.681,27.571,155.031
C02610=1066.854,105.663,426.432,172.680,27.569,155.031
C02611=1066.848,105.413,426.450,172.678,27.566,155.031
C02612=1066.842,105.164,426.469,172.677,27.563,155.030
C02613=1066.837,104.915,426.489,172.675,27.560,155.030
C02614=1066.831,104.665,426.508,172.674,27.558,155.030
C02615=1066.825,104.417,426.526,172.672,27.555,155.029
C02616=1066.819,104.167,426.545,172.671,27.552,155.029
C02617=1066.814,103.918,426.565,172.669,27.549,155.028
C02618=1066.807,103.669,426.583,172.668,27.547,155.028
C02619=1066.802,103.419,426.603,172.666,27.544,155.028
C02620=1066.797,103.171,426.621,172.665,27.541,155.027
C02621=1066.791,102.921,426.641,172.663,27.539,155.027
C02622=1066.784,102.672,426.659,172.662,27.536,155.026
C02623=1066.779,102.423,426.679,172.660,27.533,155.026
C02624=1066.773,102.173,426.698,172.659,27.530,155.026
C02625=1066.767,101.925,426.716,172.657,27.528,155.025
C02626=1066.762,101.675,426.735,172.656,27.525,155.025
C02627=1066.756,101.426,426.755,172.654,27.522,155.024
C02628=1066.749,101.177,426.773,172.653,27.519,155.024
C02629=1066.744,100.928,426.792,172.651,27.516,155.024
C02630=1066.738,100.679,426.811,172.650,27.514,155.023
C02631=1066.732,100.429,426.830,172.648,27.511,155.023
C02632=1066.726,100.180,426.849,172.647,27.509,155.023
C02633=1066.720,99.930,426.867,172.645,27.506,155.022
C02634=1066.714,99.681,426.886,172.644,27.503,155.022
C02635=1066.709,99.432,426.905,172.642,27.500,155.021
C02636=1066.703,99.183,426.923,172.641,27.497,155.021
C02637=1066.697,98.934,426.943,172.639,27.495,155.021
C02638=1066.690,98.685,426.961,172.637,27.492,155.020
C02639=1066.686,98.435,426.979,172.636,27.489,155.020
C02640=1066.679,98.186,426.998,172.634,27.487,155.019
C02641=1066.674,97.937,427.017,172.633,27.484,155.019
C02642=1066.667,97.688,427.036,172.631,27.481,155.019
C02643=1066.661,97.438,427.055,172.630,27.478,155.018
C02644=1066.656,97.189,427.073,172.628,27.476,155.018
C02645=1066.650,96.940,427.092,172.627,27.473,155.018
C02646=1066.644,96.691,427.111,172.625,27.470,155.017
C02647=1066.637,96.442,427.129,172.624,27.468,155.017
C02648=1066.633,96.192,427.147,172.622,27.465,155.016
C02649=1066.626,95.943,427.166,172.621,27.462,155.016
C02650=1066.620,95.694,427.185,172.619,27.459,155.016
C02651=1066.615,95.445,427.204,172.618,27.456,155.015
C02652=1066.609,95.195,427.222,172.616,27.454,155.015
C02653=1066.602,94.912,427.244,172.615,27.451,155.014
C02654=1066.596,94.629,427.265,172.612,27.448,155.014
C02655=1066.589,94.345,427.286,172.611,27.444,155.013
C02656=1066.582,94.062,427.307,172.609,27.442,155.013
C02657=1066.577,93.812,427.325,172.608,27.439,155.013
C02658=1066.571,93.564,427.344,172.606,27.436,155.012
C02659=1066.564,93.314,427.362,172.605,27.433,155.012
C02660=1066.559,93.064,427.381,172.603,27.430,155.011
C02661=1066.553,92.816,427.399,172.602,27.428,155.011
C02662=1066.548,92.566,427.418,172.600,27.425,155.011
C02663=1066.541,92.317,427.436,172.599,27.422,155.010
C02664=1066.535,92.068,427.455,172.597,27.420,155.010
C02665=1066.530,91.818,427.473,172.596,27.417,155.010
C02666=1066.524,91.569,427.492,172.594,27.414,155.009
C02667=1066.519,91.320,427.510,172.593,27.411,155.009
C02668=1066.512,91.071,427.529,172.591,27.409,155.008
C02669=1066.506,90.822,427.547,172.590,27.406,155.008
C02670=1066.501,90.572,427.565,172.588,27.403,155.008
C02671=1066.495,90.323,427.584,172.587,27.400,155.007
C02672=1066.489,90.073,427.602,172.585,27.398,155.007
C02673=1066.483,89.825,427.620,172.584,27.395,155.006
C02674=1066.477,89.575,427.638,172.582,27.392,155.006
C02675=1066.471,89.326,427.657,172.581,27.389,155.006
C02676=1066.466,89.077,427.675,172.579,27.387,155.005
C02677=1066.459,88.828,427.694,172.578,27.384,155.005
C02678=1066.453,88.578,427.712,172.576,27.382,155.005
C02679=1066.447,88.329,427.730,172.575,27.379,155.004
C02680=1066.441,88.080,427.748,172.573,27.376,155.004
C02681=1066.436,87.830,427.766,172.572,27.373,155.003
C02682=1066.430,87.581,427.785,172.570,27.370,155.003
C02683=1066.424,87.331,427.803,172.569,27.368,155.003
C02684=1066.417,87.082,427.821,172.567,27.365,155.002
C02685=1066.412,86.833,427.839,172.566,27.363,155.002
C02686=1066.405,86.584,427.857,172.564,27.360,155.002
C02687=1066.401,86.335,427.876,172.563,27.357,155.001
C02688=1066.394,86.085,427.894,172.561,27.354,155.001
C02689=1066.388,85.836,427.912,172.560,27.351,155.000
C02690=1066.382,85.587,427.930,172.558,27.349,155.000
C02691=1066.376,85.338,427.948,172.557,27.346,155.000
C02692=1066.371,85.089,427.966,172.555,27.343,154.999
C02693=1066.364,84.839,427.984,172.554,27.341,154.999
C02694=1066.359,84.590,428.003,172.552,27.338,154.998
C02695=1066.353,84.341,428.021,172.551,27.335,154.998
C02696=1066.347,84.091,428.039,172.550,27.332,154.998
C02697=1066.341,83.842,428.057,172.549,27.330,154.997
C02698=1066.335,83.593,428.075,172.547,27.327,154.997
C02699=1066.330,83.344,428.092,172.546,27.325,154.997
C02700=1066.323,83.094,428.111,172.544,27.322,154.996
C02701=1066.318,82.845,428.129,172.543,27.319,154.996
C02702=1066.312,82.596,428.147,172.541,27.316,154.995
C02703=1066.306,82.346,428.165,172.540,27.313,154.995
C02704=1066.300,82.097,428.183,172.538,27.311,154.995
C02705=1066.294,81.847,428.201,172.537,27.308,154.994
C02706=1066.289,81.598,428.219,172.535,27.305,154.994
C02707=1066.283,81.349,428.237,172.534,27.303,154.993
C02708=1066.277,81.100,428.255,172.532,27.300,154.993
C02709=1066.271,80.851,428.273,172.531,27.297,154.993
C02710=1066.265,80.602,428.291,172.529,27.294,154.992
C02711=1066.259,80.352,428.309,172.528,27.291,154.992
C02712=1066.253,80.103,428.327,172.526,27.289,154.991
C02713=1066.247,79.854,428.345,172.525,27.286,154.991
C02714=1066.242,79.604,428.363,172.523,27.283,154.991
C02715=1066.236,79.355,428.381,172.522,27.280,154.990
C02716=1066.231,79.105,428.398,172.520,27.278,154.990
C02717=1066.224,78.823,428.418,172.519,27.275,154.989
C02718=1066.217,78.539,428.439,172.517,27.272,154.989
C02719=1066.210,78.255,428.459,172.516,27.268,154.989
C02720=1066.203,77.972,428.479,172.513,27.265,154.988
C02721=1066.198,77.723,428.497,172.512,27.262,154.988
C02722=1066.192,77.473,428.515,172.510,27.260,154.987
C02723=1066.186,77.225,428.533,172.510,27.257,154.987
C02724=1066.180,76.975,428.551,172.508,27.255,154.987
C02725=1066.174,76.726,428.569,172.507,27.252,154.986
C02726=1066.167,76.476,428.586,172.505,27.249,154.986
C02727=1066.162,76.227,428.604,172.504,27.246,154.985
C02728=1066.156,75.978,428.622,172.502,27.244,154.985
C02729=1066.150,75.729,428.639,172.501,27.241,154.985
C02730=1066.144,75.479,428.657,172.499,27.238,154.984
C02731=1066.139,75.230,428.675,172.498,27.236,154.984
C02732=1066.132,74.980,428.693,172.496,27.233,154.984
C02733=1066.126,74.731,428.710,172.495,27.230,154.983
C02734=1066.120,74.482,428.728,172.493,27.227,154.983
C02735=1066.115,74.232,428.745,172.492,27.225,154.983
C02736=1066.109,73.983,428.763,172.490,27.222,154.982
C02737=1066.103,73.734,428.781,172.489,27.219,154.982
C02738=1066.097,73.485,428.798,172.487,27.216,154.981
C02739=1066.091,73.235,428.815,172.486,27.214,154.981
C02740=1066.085,72.986,428.833,172.484,27.211,154.981
C02741=1066.079,72.736,428.851,172.483,27.208,154.980
C02742=1066.073,72.487,428.869,172.481,27.206,154.980
C02743=1066.068,72.238,428.886,172.480,27.203,154.979
C02744=1066.062,71.989,428.904,172.479,27.200,154.979
C02745=1066.056,71.740,428.921,172.478,27.198,154.979
C02746=1066.049,71.490,428.939,172.476,27.195,154.978
C02747=1066.044,71.241,428.956,172.475,27.192,154.978
C02748=1066.039,70.991,428.973,172.473,27.190,154.978
C02749=1066.032,70.742,428.991,172.472,27.187,154.977
C02750=1066.026,70.493,429.008,172.470,27.184,154.977
C02751=1066.020,70.243,429.026,172.469,27.181,154.976
C02752=1066.015,69.994,429.044,172.467,27.178,154.976
C02753=1066.009,69.745,429.061,172.466,27.176,154.976
C02754=1066.002,69.496,429.079,172.464,27.173,154.975
C02755=1065.997,69.246,429.096,172.463,27.170,154.975
C02756=1065.991,68.996,429.113,172.461,27.168,154.974
C02757=1065.985,68.748,429.130,172.460,27.165,154.974
C02758=1065.979,68.499,429.148,172.458,27.162,154.974
C02759=1065.973,68.249,429.166,172.457,27.159,154.973
C02760=1065.967,67.999,429.182,172.455,27.157,154.973
C02761=1065.962,67.750,429.200,172.455,27.154,154.973
C02762=1065.955,67.501,429.218,172.453,27.152,154.972
C02763=1065.949,67.252,429.235,172.452,27.149,154.972
C02764=1065.943,67.002,429.252,172.450,27.146,154.971
C02765=1065.937,66.753,429.269,172.449,27.143,154.971
C02766=1065.932,66.504,429.286,172.447,27.141,154.971
C02767=1065.925,66.254,429.304,172.446,27.138,154.970
C02768=1065.920,66.005,429.321,172.445,27.135,154.970
C02769=1065.914,65.756,429.338,172.443,27.132,154.970
C02770=1065.908,65.506,429.356,172.442,27.130,154.969
C02771=1065.902,65.257,429.373,172.440,27.127,154.969
C02772=1065.896,65.008,429.390,172.439,27.124,154.968
C02773=1065.890,64.758,429.407,172.437,27.122,154.968
C02774=1065.884,64.509,429.425,172.436,27.119,154.968
C02775=1065.878,64.260,429.441,172.434,27.116,154.967
C02776=1065.872,64.010,429.459,172.433,27.114,154.967
C02777=1065.866,63.761,429.476,172.431,27.111,154.967
C02778=1065.860,63.511,429.493,172.431,27.108,154.966
C02779=1065.854,63.262,429.510,172.429,27.106,154.966
C02780=1065.848,63.013,429.526,172.428,27.103,154.965
C02781=1065.841,62.730,429.547,172.425,27.100,154.965
C02782=1065.834,62.446,429.566,172.424,27.097,154.965
C02783=1065.827,62.163,429.585,172.422,27.094,154.964
C02784=1065.820,61.879,429.605,172.421,27.091,154.964
C02785=1065.814,61.629,429.622,172.419,27.088,154.963
C02786=1065.808,61.380,429.639,172.418,27.085,154.963
C02787=1065.802,61.131,429.656,172.416,27.083,154.963
C02788=1065.796,60.881,429.673,172.415,27.080,154.962
C02789=1065.790,60.632,429.690,172.413,27.077,154.962
C02790=1065.784,60.383,429.706,172.412,27.075,154.962
C02791=1065.778,60.133,429.724,172.410,27.072,154.961
C02792=1065.772,59.884,429.740,172.409,27.070,154.961
C02793=1065.765,59.635,429.757,172.407,27.067,154.960
C02794=1065.760,59.385,429.775,172.406,27.064,154.960
C02795=1065.753,59.136,429.791,172.405,27.062,154.960
C02796=1065.748,58.886,429.808,172.404,27.059,154.959
C02797=1065.742,58.638,429.825,172.402,27.056,154.959
C02798=1065.735,58.388,429.842,172.401,27.054,154.959
C02799=1065.730,58.139,429.859,172.399,27.051,154.958
C02800=1065.724,57.889,429.876,172.398,27.048,154.958
C02801=1065.717,57.640,429.893,172.396,27.045,154.958
C02802=1065.712,57.390,429.910,172.395,27.043,154.957
C02803=1065.706,57.141,429.926,172.393,27.040,154.957
C02804=1065.700,56.892,429.943,172.392,27.038,154.956
C02805=1065.694,56.642,429.960,172.390,27.035,154.956
C02806=1065.688,56.393,429.977,172.389,27.032,154.956
C02807=1065.682,56.144,429.994,172.387,27.030,154.955
C02808=1065.676,55.894,430.010,172.386,27.027,154.955
C02809=1065.670,55.645,430.027,172.384,27.024,154.955
C02810=1065.664,55.395,430.044,172.384,27.022,154.954
C02811=1065.657,55.146,430.061,172.382,27.019,154.954
C02812=1065.652,54.897,430.078,172.381,27.016,154.953
C02813=1065.646,54.647,430.094,172.379,27.013,154.953
C02814=1065.640,54.399,430.111,172.378,27.011,154.953
C02815=1065.634,54.148,430.128,172.376,27.008,154.952
C02816=1065.628,53.899,430.145,172.375,27.006,154.952
C02817=1065.622,53.650,430.162,172.374,27.003,154.952
C02818=1065.616,53.401,430.178,172.372,27.000,154.951
C02819=1065.611,53.151,430.195,172.371,26.998,154.951
C02820=1065.604,52.902,430.212,172.369,26.995,154.951
C02821=1065.598,52.652,430.228,172.368,26.992,154.950
C02822=1065.593,52.403,430.245,172.366,26.989,154.950
C02823=1065.587,52.153,430.261,172.365,26.987,154.949
C02824=1065.580,51.905,430.278,172.364,26.984,154.949
C02825=1065.575,51.655,430.295,172.363,26.981,154.949
C02826=1065.569,51.405,430.312,172.361,26.979,154.948
C02827=1065.562,51.156,430.329,172.360,26.976,154.948
C02828=1065.557,50.907,430.345,172.358,26.973,154.948
C02829=1065.551,50.658,430.361,172.357,26.971,154.947
C02830=1065.545,50.408,430.378,172.355,26.968,154.947
C02831=1065.539,50.159,430.394,172.354,26.965,154.946
C02832=1065.533,49.910,430.411,172.352,26.962,154.946
C02833=1065.527,49.661,430.428,172.351,26.960,154.946
C02834=1065.521,49.410,430.445,172.349,26.957,154.945
C02835=1065.515,49.161,430.461,172.348,26.954,154.945
C02836=1065.509,48.911,430.477,172.346,26.951,154.945
C02837=1065.503,48.663,430.494,172.346,26.949,154.944
C02838=1065.498,48.413,430.511,172.344,26.946,154.944
C02839=1065.492,48.164,430.527,172.343,26.944,154.943
C02840=1065.486,47.914,430.544,172.341,26.941,154.943
C02841=1065.480,47.665,430.560,172.340,26.938,154.943
C02842=1065.475,47.415,430.577,172.338,26.935,154.942
C02843=1065.469,47.166,430.593,172.337,26.933,154.942
C02844=1065.463,46.917,430.610,172.335,26.930,154.942
C02845=1065.456,46.633,430.629,172.334,26.927,154.941
C02846=1065.450,46.349,430.647,172.333,26.924,154.941
C02847=1065.443,46.065,430.667,172.331,26.921,154.940
C02848=1065.436,45.781,430.685,172.329,26.917,154.940
C02849=1065.430,45.532,430.701,172.327,26.915,154.940
C02850=1065.425,45.282,430.718,172.326,26.912,154.939
C02851=1065.419,45.033,430.734,172.325,26.910,154.939
C02852=1065.413,44.784,430.750,172.324,26.907,154.938
C02853=1065.407,44.534,430.767,172.323,26.904,154.938
C02854=1065.401,44.285,430.783,172.321,26.901,154.937
C02855=1065.395,44.035,430.800,172.320,26.899,154.937
C02856=1065.390,43.786,430.816,172.318,26.896,154.937
C02857=1065.384,43.537,430.832,172.317,26.893,154.936
C02858=1065.378,43.287,430.848,172.315,26.890,154.936
C02859=1065.372,43.038,430.865,172.314,26.888,154.936
C02860=1065.366,42.789,430.881,172.312,26.885,154.935
C02861=1065.360,42.539,430.897,172.311,26.882,154.935
C02862=1065.354,42.290,430.913,172.309,26.879,154.935
C02863=1065.348,42.041,430.930,172.309,26.877,154.934
C02864=1065.342,41.791,430.946,172.307,26.875,154.934
C02865=1065.336,41.542,430.962,172.306,26.872,154.933
C02866=1065.330,41.293,430.978,172.304,26.869,154.933
C02867=1065.324,41.043,430.995,172.303,26.867,154.933
C02868=1065.318,40.794,431.011,172.301,26.864,154.932
C02869=1065.312,40.545,431.027,172.300,26.861,154.932
C02870=1065.306,40.295,431.043,172.298,26.859,154.932
C02871=1065.300,40.046,431.060,172.297,26.856,154.931
C02872=1065.294,39.797,431.076,172.295,26.853,154.931
C02873=1065.289,39.547,431.092,172.294,26.851,154.931
C02874=1065.283,39.297,431.108,172.292,26.848,154.930
C02875=1065.277,39.048,431.124,172.291,26.845,154.930
C02876=1065.271,38.798,431.140,172.290,26.842,154.929
C02877=1065.265,38.549,431.157,172.289,26.840,154.929
C02878=1065.259,38.300,431.173,172.287,26.837,154.929
C02879=1065.253,38.050,431.188,172.286,26.834,154.928
C02880=1065.247,37.801,431.204,172.285,26.832,154.928
C02881=1065.241,37.551,431.220,172.283,26.829,154.928
C02882=1065.235,37.302,431.237,172.282,26.826,154.927
C02883=1065.229,37.053,431.253,172.280,26.824,154.927
C02884=1065.223,36.803,431.268,172.279,26.821,154.927
C02885=1065.216,36.554,431.284,172.277,26.818,154.926
C02886=1065.210,36.304,431.300,172.276,26.816,154.926
C02887=1065.204,36.055,431.317,172.274,26.813,154.926
C02888=1065.199,35.805,431.332,172.273,26.810,154.925
C02889=1065.192,35.556,431.348,172.271,26.808,154.925
C02890=1065.186,35.307,431.364,172.271,26.806,154.924
C02891=1065.180,35.057,431.380,172.269,26.803,154.924
C02892=1065.175,34.807,431.396,172.268,26.800,154.924
C02893=1065.168,34.558,431.411,172.266,26.798,154.923
C02894=1065.162,34.309,431.428,172.265,26.795,154.923
C02895=1065.156,34.059,431.443,172.263,26.792,154.923
C02896=1065.150,33.810,431.459,172.262,26.790,154.922
C02897=1065.144,33.561,431.475,172.260,26.787,154.922
C02898=1065.138,33.311,431.491,172.259,26.785,154.922
C02899=1065.133,33.062,431.507,172.257,26.782,154.921
C02900=1065.127,32.813,431.523,172.256,26.779,154.921
C02901=1065.120,32.563,431.538,172.254,26.777,154.921
C02902=1065.114,32.314,431.554,172.253,26.774,154.920
C02903=1065.108,32.064,431.570,172.252,26.772,154.920
C02904=1065.103,31.814,431.586,172.251,26.769,154.920
C02905=1065.096,31.565,431.601,172.249,26.766,154.919
C02906=1065.090,31.316,431.618,172.248,26.764,154.919
C02907=1065.085,31.066,431.633,172.246,26.761,154.918
C02908=1065.079,30.817,431.650,172.245,26.758,154.918
C02909=1065.072,30.533,431.667,172.244,26.755,154.918
C02910=1065.065,30.249,431.685,172.242,26.752,154.917
C02911=1065.058,29.966,431.702,172.240,26.749,154.917
C02912=1065.051,29.682,431.720,172.238,26.746,154.917
C02913=1065.045,29.433,431.736,172.237,26.743,154.916
C02914=1065.040,29.183,431.752,172.235,26.741,154.916
C02915=1065.034,28.933,431.768,172.234,26.738,154.915
C02916=1065.028,28.684,431.783,172.232,26.735,154.915
C02917=1065.022,28.435,431.799,172.232,26.733,154.915
C02918=1065.015,28.185,431.814,172.230,26.731,154.914
C02919=1065.009,27.936,431.830,172.229,26.728,154.914
C02920=1065.004,27.686,431.846,172.227,26.725,154.914
C02921=1064.997,27.437,431.861,172.226,26.723,154.913
C02922=1064.992,27.187,431.877,172.224,26.720,154.913
C02923=1064.985,26.938,431.893,172.223,26.717,154.913
C02924=1064.980,26.689,431.908,172.221,26.715,154.912
C02925=1064.973,26.439,431.923,172.220,26.712,154.912
C02926=1064.967,26.190,431.939,172.219,26.709,154.912
C02927=1064.961,25.940,431.954,172.217,26.707,154.911
C02928=1064.955,25.691,431.970,172.216,26.704,154.911
C02929=1064.949,25.441,431.985,172.214,26.702,154.911
C02930=1064.943,25.192,432.001,172.213,26.699,154.910
C02931=1064.937,24.943,432.016,172.212,26.697,154.910
C02932=1064.931,24.693,432.032,172.211,26.694,154.910
C02933=1064.925,24.444,432.047,172.209,26.692,154.909
C02934=1064.919,24.194,432.063,172.208,26.689,154.909
C02935=1064.912,23.945,432.078,172.206,26.686,154.909
C02936=1064.907,23.695,432.094,172.205,26.684,154.908
C02937=1064.901,23.446,432.109,172.203,26.681,154.908
C02938=1064.895,23.196,432.125,172.202,26.679,154.908
C02939=1064.889,22.947,432.140,172.200,26.676,154.907
C02940=1064.883,22.697,432.155,172.199,26.674,154.907
C02941=1064.877,22.448,432.171,172.197,26.671,154.907
C02942=1064.871,22.199,432.186,172.196,26.668,154.906
C02943=1064.865,21.949,432.201,172.194,26.666,154.906
C02944=1064.859,21.699,432.217,172.193,26.663,154.905
C02945=1064.853,21.451,432.232,172.192,26.661,154.905
C02946=1064.847,21.201,432.247,172.191,26.658,154.905
C02947=1064.841,20.951,432.262,172.189,26.656,154.904
C02948=1064.835,20.702,432.279,172.188,26.653,154.904
C02949=1064.829,20.452,432.294,172.186,26.650,154.904
C02950=1064.824,20.203,432.309,172.185,26.648,154.903
C02951=1064.817,19.953,432.324,172.184,26.645,154.903
C02952=1064.811,19.704,432.339,172.182,26.642,154.903
C02953=1064.805,19.454,432.355,172.181,26.640,154.902
C02954=1064.799,19.205,432.370,172.179,26.637,154.902
C02955=1064.793,18.955,432.384,172.178,26.634,154.902
C02956=1064.787,18.706,432.401,172.176,26.632,154.901
C02957=1064.780,18.456,432.416,172.175,26.629,154.901
C02958=1064.775,18.207,432.430,172.173,26.627,154.901
C02959=1064.769,17.957,432.446,172.173,26.624,154.900
C02960=1064.763,17.708,432.461,172.171,26.622,154.900
C02961=1064.756,17.458,432.476,172.170,26.619,154.900
C02962=1064.751,17.209,432.492,172.168,26.617,154.899
C02963=1064.745,16.960,432.507,172.167,26.614,154.899
C02964=1064.738,16.710,432.521,172.165,26.612,154.899
C02965=1064.733,16.461,432.537,172.164,26.609,154.898
C02966=1064.727,16.211,432.552,172.162,26.607,154.898
C02967=1064.720,15.962,432.567,172.161,26.604,154.898
C02968=1064.715,15.712,432.582,172.159,26.601,154.897
C02969=1064.709,15.463,432.597,172.158,26.599,154.897
C02970=1064.702,15.214,432.612,172.156,26.596,154.897
C02971=1064.697,14.964,432.628,172.155,26.593,154.896
C02972=1064.691,14.715,432.642,172.153,26.591,154.896
C02973=1064.683,14.432,432.660,172.152,26.588,154.896
C02974=1064.677,14.150,432.676,172.150,26.585,154.895
C02975=1064.671,13.867,432.694,172.149,26.583,154.895
C02976=1064.663,13.584,432.711,172.148,26.580,154.895
C02977=1064.657,13.335,432.725,172.146,26.577,154.894
C02978=1064.651,13.086,432.740,172.145,26.575,154.894
C02979=1064.645,12.836,432.755,172.143,26.572,154.894
C02980=1064.638,12.586,432.770,172.142,26.570,154.893
C02981=1064.632,12.338,432.785,172.140,26.567,154.893
C02982=1064.626,12.088,432.800,172.139,26.565,154.893
C02983=1064.620,11.838,432.814,172.137,26.562,154.892
C02984=1064.614,11.589,432.829,172.136,26.560,154.892
C02985=1064.608,11.339,432.845,172.134,26.557,154.892
C02986=1064.602,11.090,432.860,172.133,26.555,154.891
C02987=1064.596,10.841,432.874,172.131,26.552,154.891
C02988=1064.590,10.591,432.889,172.130,26.550,154.891
C02989=1064.583,10.341,432.904,172.128,26.547,154.890
C02990=1064.578,10.092,432.918,172.127,26.545,154.890
C02991=1064.571,9.842,432.933,172.125,26.542,154.890
C02992=1064.565,9.592,432.948,172.125,26.540,154.889
C02993=1064.559,9.344,432.962,172.123,26.537,154.889
C02994=1064.553,9.094,432.977,172.122,26.535,154.889
C02995=1064.547,8.844,432.992,172.120,26.532,154.888
C02996=1064.541,8.595,433.007,172.119,26.530,154.888
C02997=1064.534,8.346,433.022,172.117,26.527,154.888
C02998=1064.529,8.096,433.037,172.116,26.525,154.888
C02999=1064.523,7.846,433.051,172.114,26.523,154.887
C03000=1064.517,7.596,433.066,172.113,26.520,154.887
C03001=1064.511,7.347,433.081,172.111,26.517,154.887
C03002=1064.505,7.098,433.096,172.110,26.515,154.886
C03003=1064.498,6.848,433.111,172.108,26.512,154.886
C03004=1064.493,6.599,433.125,172.107,26.510,154.886
C03005=1064.486,6.349,433.139,172.105,26.507,154.885
C03006=1064.481,6.100,433.154,172.104,26.505,154.885
C03007=1064.474,5.850,433.169,172.102,26.502,154.885
C03008=1064.468,5.601,433.184,172.101,26.500,154.884
C03009=1064.462,5.352,433.198,172.099,26.497,154.884
C03010=1064.456,5.101,433.213,172.098,26.495,154.884
C03011=1064.450,4.852,433.227,172.097,26.492,154.883
C03012=1064.444,4.603,433.242,172.096,26.490,154.883
C03013=1064.438,4.354,433.257,172.094,26.488,154.883
C03014=1064.432,4.104,433.271,172.093,26.485,154.882
C03015=1064.426,3.855,433.286,172.091,26.483,154.882
C03016=1064.420,3.605,433.301,172.090,26.480,154.882
C03017=1064.414,3.356,433.315,172.088,26.477,154.882
C03018=1064.408,3.106,433.329,172.087,26.475,154.881
C03019=1064.402,2.856,433.344,172.086,26.472,154.881
C03020=1064.396,2.607,433.359,172.084,26.470,154.881
C03021=1064.390,2.357,433.373,172.082,26.468,154.880
C03022=1064.384,2.108,433.388,172.081,26.465,154.880
C03023=1064.378,1.858,433.403,172.080,26.462,154.880
C03024=1064.372,1.609,433.417,172.078,26.460,154.879
C03025=1064.366,1.359,433.431,172.077,26.457,154.879
C03026=1064.360,1.110,433.446,172.075,26.455,154.879
C03027=1064.354,0.860,433.460,172.074,26.452,154.878
C03028=1064.348,0.611,433.475,172.072,26.450,154.878
C03029=1064.342,0.362,433.489,172.071,26.447,154.878
C03030=1064.336,0.112,433.504,172.069,26.445,154.877
C03031=1064.330,-0.137,433.518,172.069,26.443,154.877
C03032=1064.324,-0.388,433.532,172.067,26.440,154.877
C03033=1064.319,-0.637,433.547,172.066,26.437,154.876
C03034=1064.312,-0.886,433.562,172.064,26.435,154.876
C03035=1064.307,-1.136,433.576,172.063,26.433,154.876
C03036=1064.300,-1.386,433.591,172.061,26.430,154.876
C03037=1064.294,-1.666,433.606,172.060,26.428,154.875
C03038=1064.287,-1.946,433.623,172.057,26.424,154.875
C03039=1064.281,-2.226,433.639,172.056,26.421,154.875
C03040=1064.274,-2.508,433.655,172.055,26.419,154.874
C03041=1064.268,-2.757,433.670,172.053,26.416,154.874
C03042=1064.262,-3.007,433.684,172.051,26.414,154.874
C03043=1064.256,-3.256,433.698,172.050,26.411,154.873
C03044=1064.250,-3.506,433.712,172.049,26.409,154.873
C03045=1064.244,-3.755,433.727,172.047,26.407,154.873
C03046=1064.238,-4.005,433.741,172.046,26.404,154.872
C03047=1064.232,-4.254,433.755,172.044,26.402,154.872
C03048=1064.225,-4.504,433.769,172.043,26.399,154.872
C03049=1064.219,-4.753,433.784,172.041,26.397,154.871
C03050=1064.213,-5.003,433.798,172.040,26.394,154.871
C03051=1064.207,-5.252,433.812,172.038,26.392,154.871
C03052=1064.201,-5.501,433.826,172.036,26.390,154.871
C03053=1064.195,-5.752,433.840,172.035,26.387,154.870
C03054=1064.189,-6.000,433.854,172.035,26.385,154.870
C03055=1064.183,-6.251,433.868,172.033,26.383,154.870
C03056=1064.177,-6.499,433.883,172.031,26.380,154.869
C03057=1064.170,-6.749,433.896,172.030,26.378,154.869
C03058=1064.164,-6.999,433.910,172.028,26.376,154.869
C03059=1064.159,-7.248,433.925,172.027,26.373,154.869
C03060=1064.152,-7.498,433.939,172.026,26.370,154.868
C03061=1064.146,-7.747,433.953,172.024,26.368,154.868
C03062=1064.140,-7.997,433.967,172.022,26.366,154.868
C03063=1064.134,-8.246,433.981,172.021,26.364,154.867
C03064=1064.127,-8.496,433.996,172.019,26.361,154.867
C03065=1064.122,-8.746,434.009,172.018,26.359,154.867
C03066=1064.116,-8.995,434.023,172.017,26.356,154.867
C03067=1064.109,-9.245,434.038,172.015,26.354,154.866
C03068=1064.104,-9.494,434.051,172.013,26.351,154.866
C03069=1064.098,-9.743,434.065,172.012,26.349,154.866
C03070=1064.091,-9.993,434.080,172.010,26.347,154.865
C03071=1064.086,-10.243,434.094,172.009,26.344,154.865
C03072=1064.079,-10.493,434.107,172.008,26.342,154.865
C03073=1064.074,-10.742,434.121,172.006,26.339,154.865
C03074=1064.067,-10.991,434.135,172.004,26.337,154.864
C03075=1064.061,-11.241,434.149,172.003,26.335,154.864
C03076=1064.055,-11.491,434.163,172.001,26.332,154.864
C03077=1064.049,-11.740,434.176,172.000,26.330,154.863
C03078=1064.043,-11.990,434.191,171.998,26.328,154.863
C03079=1064.037,-12.239,434.205,171.997,26.325,154.863
C03080=1064.031,-12.488,434.218,171.996,26.322,154.863
C03081=1064.025,-12.739,434.233,171.994,26.320,154.862
C03082=1064.019,-12.987,434.247,171.992,26.318,154.862
C03083=1064.013,-13.237,434.261,171.991,26.316,154.862
C03084=1064.008,-13.487,434.274,171.989,26.313,154.861
C03085=1064.001,-13.737,434.288,171.988,26.311,154.861
C03086=1063.995,-13.986,434.302,171.986,26.309,154.861
C03087=1063.989,-14.235,434.315,171.986,26.306,154.860
C03088=1063.983,-14.485,434.330,171.984,26.304,154.860
C03089=1063.977,-14.735,434.344,171.983,26.301,154.860
C03090=1063.971,-14.984,434.357,171.981,26.299,154.860
C03091=1063.965,-15.234,434.372,171.980,26.297,154.859
C03092=1063.959,-15.483,434.385,171.978,26.294,154.859
C03093=1063.953,-15.733,434.398,171.977,26.292,154.859
C03094=1063.947,-15.982,434.412,171.975,26.290,154.859
C03095=1063.940,-16.232,434.426,171.974,26.287,154.858
C03096=1063.935,-16.482,434.439,171.972,26.285,154.858
C03097=1063.928,-16.730,434.453,171.971,26.283,154.858
C03098=1063.921,-16.980,434.467,171.969,26.281,154.858
C03099=1063.916,-17.230,434.481,171.968,26.278,154.857
C03100=1063.910,-17.479,434.494,171.966,26.276,154.857
C03101=1063.902,-17.759,434.510,171.965,26.274,154.857
C03102=1063.896,-18.037,434.525,171.962,26.271,154.856
C03103=1063.889,-18.316,434.540,171.961,26.268,154.856
C03104=1063.882,-18.595,434.555,171.959,26.266,154.856
C03105=1063.877,-18.844,434.569,171.958,26.263,154.856
C03106=1063.870,-19.094,434.583,171.956,26.261,154.855
C03107=1063.864,-19.344,434.596,171.955,26.259,154.855
C03108=1063.858,-19.593,434.610,171.953,26.256,154.855
C03109=1063.852,-19.843,434.623,171.952,26.254,154.855
C03110=1063.846,-20.093,434.637,171.950,26.252,154.854
C03111=1063.840,-20.342,434.650,171.949,26.250,154.854
C03112=1063.833,-20.591,434.664,171.947,26.247,154.854
C03113=1063.828,-20.841,434.678,171.946,26.245,154.853
C03114=1063.822,-21.090,434.691,171.944,26.243,154.853
C03115=1063.815,-21.341,434.704,171.943,26.240,154.853
C03116=1063.810,-21.590,434.718,171.941,26.238,154.853
C03117=1063.803,-21.840,434.731,171.940,26.236,154.852
C03118=1063.797,-22.089,434.744,171.938,26.233,154.852
C03119=1063.791,-22.339,434.758,171.937,26.232,154.852
C03120=1063.785,-22.588,434.772,171.935,26.229,154.852
C03121=1063.779,-22.838,434.785,171.934,26.227,154.851
C03122=1063.773,-23.087,434.799,171.932,26.225,154.851
C03123=1063.767,-23.337,434.812,171.931,26.222,154.851
C03124=1063.761,-23.586,434.825,171.929,26.220,154.851
C03125=1063.755,-23.837,434.839,171.928,26.218,154.850
C03126=1063.749,-24.086,434.852,171.926,26.215,154.850
C03127=1063.743,-24.335,434.865,171.925,26.213,154.850
C03128=1063.737,-24.585,434.879,171.923,26.211,154.850
C03129=1063.731,-24.834,434.893,171.922,26.208,154.849
C03130=1063.725,-25.083,434.906,171.920,26.206,154.849
C03131=1063.719,-25.334,434.919,171.919,26.204,154.849
C03132=1063.713,-25.583,434.933,171.917,26.201,154.848
C03133=1063.707,-25.833,434.946,171.915,26.200,154.848
C03134=1063.701,-26.082,434.960,171.914,26.197,154.848
C03135=1063.695,-26.332,434.973,171.912,26.195,154.848
C03136=1063.689,-26.581,434.986,171.911,26.193,154.848
C03137=1063.683,-26.831,434.999,171.909,26.190,154.847
C03138=1063.676,-27.080,435.012,171.908,26.188,154.847
C03139=1063.670,-27.330,435.026,171.906,26.186,154.847
C03140=1063.664,-27.580,435.039,171.905,26.184,154.847
C03141=1063.658,-27.829,435.052,171.903,26.182,154.846
C03142=1063.652,-28.079,435.065,171.902,26.179,154.846
C03143=1063.646,-28.328,435.079,171.900,26.177,154.846
C03144=1063.640,-28.578,435.091,171.899,26.175,154.846
C03145=1063.633,-28.828,435.105,171.897,26.173,154.845
C03146=1063.627,-29.077,435.118,171.896,26.171,154.845
C03147=1063.621,-29.327,435.131,171.894,26.168,154.845
C03148=1063.615,-29.576,435.144,171.893,26.166,154.845
C03149=1063.609,-29.826,435.158,171.891,26.164,154.844
C03150=1063.603,-30.076,435.170,171.889,26.162,154.844
C03151=1063.597,-30.325,435.184,171.888,26.160,154.844
C03152=1063.591,-30.574,435.197,171.886,26.157,154.844
C03153=1063.584,-30.825,435.210,171.885,26.155,154.843
C03154=1063.578,-31.074,435.223,171.883,26.153,154.843
C03155=1063.572,-31.323,435.236,171.882,26.151,154.843
C03156=1063.566,-31.573,435.249,171.880,26.149,154.843
C03157=1063.560,-31.822,435.262,171.879,26.147,154.843
C03158=1063.554,-32.072,435.275,171.877,26.144,154.842
C03159=1063.548,-32.322,435.288,171.876,26.142,154.842
C03160=1063.542,-32.571,435.301,171.874,26.140,154.842
C03161=1063.536,-32.821,435.314,171.873,26.138,154.842
C03162=1063.529,-33.070,435.327,171.871,26.136,154.841
C03163=1063.524,-33.320,435.340,171.870,26.133,154.841
C03164=1063.517,-33.569,435.353,171.868,26.132,154.841
C03165=1063.511,-33.848,435.368,171.866,26.129,154.841
C03166=1063.504,-34.126,435.382,171.865,26.127,154.840
C03167=1063.497,-34.404,435.397,171.862,26.124,154.840
C03168=1063.490,-34.682,435.412,171.861,26.122,154.840
C03169=1063.484,-34.932,435.424,171.859,26.120,154.840
C03170=1063.478,-35.181,435.437,171.858,26.117,154.839
C03171=1063.472,-35.431,435.450,171.856,26.116,154.839
C03172=1063.466,-35.680,435.463,171.855,26.113,154.839
C03173=1063.460,-35.930,435.476,171.853,26.111,154.839
C03174=1063.454,-36.180,435.488,171.852,26.109,154.838
C03175=1063.448,-36.429,435.502,171.850,26.107,154.838
C03176=1063.442,-36.679,435.514,171.849,26.105,154.838
C03177=1063.436,-36.929,435.527,171.847,26.102,154.838
C03178=1063.430,-37.178,435.540,171.846,26.100,154.838
C03179=1063.423,-37.428,435.553,171.844,26.098,154.837
C03180=1063.418,-37.678,435.566,171.843,26.096,154.837
C03181=1063.411,-37.927,435.579,171.841,26.094,154.837
C03182=1063.406,-38.176,435.591,171.839,26.092,154.837
C03183=1063.400,-38.426,435.604,171.838,26.089,154.836
C03184=1063.394,-38.675,435.617,171.836,26.088,154.836
C03185=1063.388,-38.925,435.630,171.835,26.085,154.836
C03186=1063.382,-39.174,435.643,171.833,26.084,154.836
C03187=1063.375,-39.424,435.655,171.832,26.081,154.836
C03188=1063.369,-39.674,435.667,171.830,26.080,154.835
C03189=1063.363,-39.923,435.681,171.829,26.077,154.835
C03190=1063.357,-40.173,435.693,171.827,26.075,154.835
C03191=1063.351,-40.423,435.706,171.825,26.073,154.835
C03192=1063.344,-40.672,435.718,171.824,26.071,154.835
C03193=1063.338,-40.922,435.731,171.822,26.069,154.834
C03194=1063.332,-41.171,435.744,171.821,26.067,154.834
C03195=1063.326,-41.421,435.757,171.819,26.065,154.834
C03196=1063.320,-41.671,435.769,171.818,26.063,154.834
C03197=1063.314,-41.920,435.781,171.816,26.061,154.834
C03198=1063.308,-42.170,435.794,171.814,26.059,154.833
C03199=1063.302,-42.419,435.807,171.813,26.057,154.833
C03200=1063.296,-42.669,435.820,171.811,26.055,154.833
C03201=1063.289,-42.919,435.832,171.810,26.053,154.833
C03202=1063.283,-43.169,435.844,171.808,26.051,154.833
C03203=1063.277,-43.418,435.857,171.807,26.049,154.832
C03204=1063.271,-43.668,435.870,171.805,26.047,154.832
C03205=1063.265,-43.918,435.883,171.804,26.044,154.832
C03206=1063.258,-44.167,435.895,171.802,26.043,154.832
C03207=1063.252,-44.417,435.908,171.801,26.040,154.832
C03208=1063.247,-44.666,435.920,171.798,26.038,154.831
C03209=1063.241,-44.916,435.933,171.796,26.036,154.831
C03210=1063.234,-45.165,435.944,171.795,26.034,154.831
C03211=1063.228,-45.415,435.957,171.793,26.032,154.831
C03212=1063.222,-45.664,435.970,171.792,26.030,154.831
C03213=1063.216,-45.914,435.982,171.790,26.028,154.830
C03214=1063.210,-46.164,435.995,171.789,26.026,154.830
C03215=1063.204,-46.414,436.007,171.787,26.024,154.830
C03216=1063.198,-46.664,436.020,171.786,26.022,154.830
C03217=1063.192,-46.912,436.032,171.784,26.020,154.830
C03218=1063.186,-47.162,436.044,171.782,26.018,154.829
C03219=1063.180,-47.412,436.057,171.781,26.016,154.829
C03220=1063.174,-47.661,436.070,171.779,26.014,154.829
C03221=1063.167,-47.911,436.082,171.778,26.012,154.829
C03222=1063.161,-48.161,436.094,171.776,26.010,154.829
C03223=1063.156,-48.410,436.107,171.775,26.008,154.828
C03224=1063.149,-48.660,436.119,171.773,26.006,154.828
C03225=1063.143,-48.910,436.131,171.771,26.004,154.828
C03226=1063.137,-49.159,436.144,171.770,26.002,154.828
C03227=1063.131,-49.409,436.156,171.768,26.000,154.828
C03228=1063.125,-49.659,436.168,171.767,25.998,154.827
C03229=1063.118,-49.937,436.182,171.765,25.996,154.827
C03230=1063.111,-50.215,436.196,171.763,25.994,154.827
C03231=1063.104,-50.494,436.210,171.761,25.991,154.827
C03232=1063.098,-50.772,436.223,171.760,25.990,154.827
C03233=1063.092,-51.022,436.236,171.758,25.988,154.827
C03234=1063.085,-51.272,436.248,171.756,25.985,154.826
C03235=1063.079,-51.522,436.260,171.755,25.984,154.826
C03236=1063.073,-51.771,436.272,171.753,25.982,154.826
C03237=1063.066,-52.020,436.284,171.752,25.980,154.826
C03238=1063.060,-52.270,436.296,171.750,25.978,154.826
C03239=1063.054,-52.520,436.308,171.749,25.976,154.825
C03240=1063.048,-52.769,436.321,171.747,25.974,154.825
C03241=1063.041,-53.019,436.333,171.745,25.973,154.825
C03242=1063.035,-53.269,436.344,171.744,25.971,154.825
C03243=1063.030,-53.518,436.356,171.741,25.969,154.825
C03244=1063.023,-53.768,436.368,171.740,25.967,154.825
C03245=1063.017,-54.018,436.381,171.738,25.965,154.825
C03246=1063.010,-54.267,436.393,171.736,25.963,154.824
C03247=1063.004,-54.517,436.405,171.735,25.961,154.824
C03248=1062.998,-54.766,436.417,171.733,25.959,154.824
C03249=1062.992,-55.016,436.429,171.732,25.958,154.824
C03250=1062.986,-55.266,436.441,171.730,25.956,154.824
C03251=1062.980,-55.516,436.453,171.728,25.954,154.824
C03252=1062.973,-55.765,436.464,171.727,25.952,154.823
C03253=1062.968,-56.015,436.477,171.725,25.950,154.823
C03254=1062.961,-56.264,436.489,171.724,25.948,154.823
C03255=1062.954,-56.514,436.501,171.722,25.946,154.823
C03256=1062.948,-56.764,436.513,171.720,25.945,154.823
C03257=1062.942,-57.014,436.524,171.719,25.943,154.823
C03258=1062.936,-57.263,436.536,171.717,25.941,154.823
C03259=1062.930,-57.513,436.549,171.716,25.939,154.822
C03260=1062.923,-57.762,436.560,171.714,25.937,154.822
C03261=1062.917,-58.012,436.572,171.712,25.935,154.822
C03262=1062.912,-58.262,436.584,171.711,25.934,154.822
C03263=1062.905,-58.511,436.596,171.709,25.932,154.822
C03264=1062.899,-58.761,436.608,171.708,25.930,154.822
C03265=1062.893,-59.011,436.620,171.706,25.928,154.821
C03266=1062.887,-59.260,436.631,171.704,25.927,154.821
C03267=1062.881,-59.510,436.644,171.703,25.925,154.821
C03268=1062.874,-59.759,436.656,171.700,25.923,154.821
C03269=1062.868,-60.008,436.667,171.699,25.921,154.821
C03270=1062.862,-60.259,436.679,171.697,25.919,154.821
C03271=1062.856,-60.508,436.691,171.695,25.917,154.821
C03272=1062.850,-60.757,436.703,171.694,25.916,154.820
C03273=1062.844,-61.008,436.714,171.692,25.914,154.820
C03274=1062.838,-61.257,436.727,171.691,25.912,154.820
C03275=1062.831,-61.507,436.739,171.689,25.910,154.820
C03276=1062.825,-61.756,436.750,171.687,25.908,154.820
C03277=1062.819,-62.006,436.762,171.686,25.906,154.820
C03278=1062.813,-62.256,436.774,171.684,25.904,154.819
C03279=1062.807,-62.505,436.785,171.683,25.903,154.819
C03280=1062.801,-62.755,436.797,171.681,25.901,154.819
C03281=1062.794,-63.005,436.809,171.679,25.899,154.819
C03282=1062.789,-63.254,436.820,171.678,25.897,154.819
C03283=1062.782,-63.504,436.832,171.676,25.896,154.819
C03284=1062.777,-63.753,436.844,171.675,25.894,154.819
C03285=1062.770,-64.003,436.856,171.673,25.892,154.818
C03286=1062.764,-64.253,436.868,171.671,25.890,154.818
C03287=1062.759,-64.503,436.879,171.670,25.889,154.818
C03288=1062.752,-64.752,436.891,171.668,25.887,154.818
C03289=1062.746,-65.002,436.903,171.666,25.885,154.818
C03290=1062.740,-65.251,436.914,171.665,25.883,154.818
C03291=1062.734,-65.501,436.926,171.662,25.881,154.818
C03292=1062.728,-65.751,436.937,171.661,25.879,154.818
C03293=1062.721,-66.030,436.950,171.659,25.878,154.817
C03294=1062.714,-66.310,436.963,171.658,25.876,154.817
C03295=1062.707,-66.590,436.977,171.656,25.874,154.817
C03296=1062.701,-66.869,436.990,171.653,25.872,154.817
C03297=1062.694,-67.120,437.001,171.652,25.870,154.817
C03298=1062.688,-67.369,437.013,171.650,25.869,154.817
C03299=1062.683,-67.619,437.024,171.649,25.867,154.817
C03300=1062.676,-67.869,437.036,171.647,25.865,154.816
C03301=1062.670,-68.118,437.047,171.645,25.863,154.816
C03302=1062.665,-68.369,437.059,171.644,25.862,154.816
C03303=1062.659,-68.617,437.071,171.642,25.860,154.816
C03304=1062.652,-68.868,437.082,171.640,25.858,154.816
C03305=1062.646,-69.116,437.093,171.639,25.856,154.816
C03306=1062.641,-69.367,437.105,171.637,25.854,154.816
C03307=1062.634,-69.616,437.117,171.636,25.853,154.815
C03308=1062.628,-69.866,437.128,171.634,25.852,154.815
C03309=1062.622,-70.115,437.140,171.632,25.850,154.815
C03310=1062.616,-70.365,437.151,171.631,25.848,154.815
C03311=1062.611,-70.615,437.162,171.629,25.846,154.815
C03312=1062.604,-70.864,437.174,171.627,25.844,154.815
C03313=1062.598,-71.114,437.185,171.625,25.842,154.815
C03314=1062.592,-71.364,437.197,171.623,25.841,154.815
C03315=1062.587,-71.613,437.209,171.622,25.839,154.815
C03316=1062.580,-71.864,437.220,171.620,25.838,154.814
C03317=1062.574,-72.112,437.231,171.618,25.836,154.814
C03318=1062.568,-72.363,437.243,171.617,25.834,154.814
C03319=1062.562,-72.612,437.254,171.615,25.832,154.814
C03320=1062.556,-72.862,437.266,171.614,25.831,154.814
C03321=1062.551,-73.111,437.277,171.612,25.829,154.814
C03322=1062.544,-73.362,437.288,171.610,25.827,154.814
C03323=1062.538,-73.610,437.300,171.609,25.826,154.814
C03324=1062.532,-73.861,437.311,171.607,25.824,154.813
C03325=1062.526,-74.110,437.322,171.605,25.822,154.813
C03326=1062.520,-74.360,437.333,171.604,25.821,154.813
C03327=1062.514,-74.609,437.345,171.602,25.819,154.813
C03328=1062.507,-74.859,437.356,171.600,25.818,154.813
C03329=1062.502,-75.109,437.367,171.599,25.816,154.813
C03330=1062.495,-75.358,437.379,171.597,25.815,154.813
C03331=1062.489,-75.608,437.390,171.595,25.813,154.813
C03332=1062.483,-75.858,437.401,171.594,25.811,154.813
C03333=1062.477,-76.108,437.412,171.591,25.810,154.813
C03334=1062.471,-76.357,437.423,171.590,25.808,154.812
C03335=1062.465,-76.607,437.435,171.588,25.806,154.812
C03336=1062.459,-76.856,437.446,171.586,25.805,154.812
C03337=1062.453,-77.106,437.457,171.585,25.803,154.812
C03338=1062.447,-77.356,437.468,171.583,25.802,154.812
C03339=1062.441,-77.606,437.479,171.581,25.800,154.812
C03340=1062.435,-77.855,437.491,171.580,25.798,154.812
C03341=1062.428,-78.105,437.502,171.578,25.797,154.812
C03342=1062.423,-78.355,437.513,171.576,25.795,154.812
C03343=1062.416,-78.604,437.523,171.575,25.794,154.812
C03344=1062.410,-78.854,437.534,171.573,25.792,154.812
C03345=1062.404,-79.103,437.545,171.571,25.791,154.811
C03346=1062.398,-79.354,437.556,171.570,25.790,154.811
C03347=1062.392,-79.603,437.568,171.568,25.788,154.811
C03348=1062.385,-79.853,437.579,171.566,25.787,154.811
C03349=1062.380,-80.102,437.590,171.565,25.785,154.811
C03350=1062.373,-80.352,437.601,171.563,25.784,154.811
C03351=1062.367,-80.602,437.612,171.561,25.782,154.811
C03352=1062.361,-80.851,437.622,171.559,25.780,154.811
C03353=1062.355,-81.101,437.634,171.557,25.779,154.811
C03354=1062.348,-81.350,437.644,171.555,25.777,154.811
C03355=1062.342,-81.601,437.655,171.554,25.776,154.811
C03356=1062.336,-81.850,437.666,171.552,25.774,154.811
C03357=1062.329,-82.133,437.679,171.550,25.773,154.811
C03358=1062.322,-82.414,437.691,171.549,25.771,154.810
C03359=1062.315,-82.696,437.703,171.546,25.769,154.810
C03360=1062.308,-82.978,437.716,171.544,25.768,154.810
C03361=1062.302,-83.228,437.726,171.543,25.766,154.810
C03362=1062.295,-83.478,437.737,171.541,25.765,154.810
C03363=1062.290,-83.727,437.748,171.539,25.764,154.810
C03364=1062.283,-83.977,437.758,171.538,25.762,154.810
C03365=1062.277,-84.227,437.770,171.536,25.761,154.810
C03366=1062.271,-84.476,437.780,171.534,25.760,154.810
C03367=1062.264,-84.726,437.791,171.533,25.758,154.810
C03368=1062.258,-84.976,437.802,171.530,25.757,154.810
C03369=1062.252,-85.225,437.813,171.528,25.755,154.810
C03370=1062.245,-85.475,437.823,171.527,25.754,154.810
C03371=1062.240,-85.724,437.834,171.525,25.752,154.810
C03372=1062.234,-85.974,437.845,171.523,25.751,154.810
C03373=1062.228,-86.224,437.856,171.522,25.750,154.810
C03374=1062.221,-86.473,437.867,171.520,25.748,154.810
C03375=1062.216,-86.723,437.877,171.518,25.747,154.809
C03376=1062.209,-86.974,437.888,171.517,25.745,154.809
C03377=1062.203,-87.223,437.898,171.515,25.744,154.809
C03378=1062.197,-87.472,437.909,171.513,25.743,154.809
C03379=1062.191,-87.722,437.921,171.512,25.741,154.809
C03380=1062.184,-87.972,437.931,171.510,25.740,154.809
C03381=1062.178,-88.221,437.942,171.508,25.739,154.809
C03382=1062.171,-88.471,437.952,171.506,25.737,154.809
C03383=1062.166,-88.721,437.963,171.505,25.736,154.809
C03384=1062.160,-88.971,437.973,171.503,25.735,154.809
C03385=1062.153,-89.220,437.984,171.501,25.734,154.809
C03386=1062.147,-89.470,437.995,171.499,25.731,154.809
C03387=1062.142,-89.719,438.006,171.497,25.730,154.809
C03388=1062.135,-89.969,438.015,171.495,25.729,154.809
C03389=1062.129,-90.219,438.027,171.494,25.728,154.809
C03390=1062.123,-90.469,438.037,171.492,25.726,154.809
C03391=1062.117,-90.718,438.048,171.490,25.725,154.809
C03392=1062.111,-90.968,438.059,171.488,25.724,154.809
C03393=1062.104,-91.218,438.069,171.487,25.723,154.809
C03394=1062.099,-91.468,438.079,171.485,25.721,154.808
C03395=1062.093,-91.717,438.090,171.483,25.720,154.808
C03396=1062.086,-91.966,438.101,171.482,25.718,154.808
C03397=1062.080,-92.217,438.111,171.480,25.717,154.808
C03398=1062.075,-92.467,438.122,171.478,25.716,154.808
C03399=1062.068,-92.716,438.132,171.477,25.714,154.808
C03400=1062.063,-92.966,438.142,171.475,25.713,154.808
C03401=1062.056,-93.216,438.153,171.473,25.712,154.808
C03402=1062.050,-93.465,438.164,171.471,25.711,154.808
C03403=1062.044,-93.715,438.175,171.470,25.709,154.808
C03404=1062.038,-93.965,438.184,171.468,25.708,154.808
C03405=1062.032,-94.214,438.195,171.465,25.706,154.808
C03406=1062.025,-94.464,438.206,171.464,25.705,154.808
C03407=1062.020,-94.714,438.216,171.462,25.704,154.808
C03408=1062.013,-94.963,438.226,171.460,25.703,154.808
C03409=1062.008,-95.213,438.237,171.459,25.701,154.808
C03410=1062.002,-95.463,438.247,171.457,25.700,154.808
C03411=1061.995,-95.713,438.258,171.455,25.699,154.808
C03412=1061.990,-95.963,438.268,171.453,25.697,154.808
C03413=1061.983,-96.212,438.279,171.452,25.696,154.808
C03414=1061.977,-96.461,438.289,171.450,25.695,154.808
C03415=1061.971,-96.711,438.299,171.448,25.694,154.808
C03416=1061.966,-96.961,438.310,171.447,25.692,154.808
C03417=1061.960,-97.211,438.320,171.445,25.691,154.808
C03418=1061.953,-97.461,438.331,171.443,25.690,154.808
C03419=1061.947,-97.710,438.342,171.441,25.689,154.808
C03420=1061.941,-97.960,438.351,171.440,25.688,154.808
C03421=1061.934,-98.244,438.362,171.437,25.686,154.808
C03422=1061.927,-98.529,438.374,171.435,25.685,154.808
C03423=1061.920,-98.813,438.385,171.433,25.684,154.808
C03424=1061.913,-99.097,438.397,171.431,25.682,154.808
C03425=1061.907,-99.346,438.408,171.429,25.681,154.808
C03426=1061.900,-99.597,438.419,171.427,25.680,154.808
C03427=1061.894,-99.846,438.428,171.426,25.679,154.808
C03428=1061.888,-100.096,438.439,171.424,25.678,154.808
C03429=1061.882,-100.346,438.449,171.422,25.676,154.808
C03430=1061.876,-100.595,438.458,171.420,25.675,154.808
C03431=1061.870,-100.845,438.469,171.419,25.674,154.808
C03432=1061.864,-101.095,438.479,171.417,25.673,154.808
C03433=1061.857,-101.345,438.489,171.415,25.672,154.808
C03434=1061.851,-101.594,438.499,171.413,25.671,154.808
C03435=1061.845,-101.844,438.510,171.412,25.670,154.808
C03436=1061.839,-102.094,438.520,171.410,25.669,154.808
C03437=1061.833,-102.343,438.530,171.408,25.667,154.808
C03438=1061.827,-102.593,438.540,171.406,25.666,154.808
C03439=1061.821,-102.843,438.550,171.405,25.665,154.808
C03440=1061.815,-103.092,438.560,171.402,25.664,154.808
C03441=1061.809,-103.343,438.570,171.400,25.663,154.808
C03442=1061.802,-103.592,438.581,171.399,25.662,154.808
C03443=1061.796,-103.842,438.590,171.397,25.661,154.808
C03444=1061.790,-104.092,438.600,171.395,25.659,154.808
C03445=1061.784,-104.341,438.611,171.393,25.658,154.808
C03446=1061.778,-104.591,438.620,171.391,25.658,154.808
C03447=1061.772,-104.841,438.630,171.390,25.656,154.808
C03448=1061.766,-105.090,438.641,171.388,25.655,154.808
C03449=1061.760,-105.340,438.650,171.386,25.654,154.808
C03450=1061.754,-105.590,438.660,171.385,25.653,154.808
C03451=1061.747,-105.839,438.670,171.383,25.652,154.808
C03452=1061.742,-106.089,438.680,171.381,25.651,154.808
C03453=1061.735,-106.339,438.690,171.379,25.650,154.808
C03454=1061.729,-106.588,438.700,171.377,25.649,154.808
C03455=1061.723,-106.838,438.710,171.376,25.648,154.808
C03456=1061.717,-107.089,438.720,171.374,25.647,154.808
C03457=1061.711,-107.338,438.730,171.372,25.646,154.808
C03458=1061.704,-107.588,438.740,171.370,25.645,154.808
C03459=1061.698,-107.837,438.750,171.369,25.644,154.808
C03460=1061.692,-108.087,438.759,171.366,25.642,154.808
C03461=1061.686,-108.337,438.769,171.364,25.642,154.808
C03462=1061.679,-108.586,438.779,171.362,25.640,154.808
C03463=1061.674,-108.836,438.789,171.361,25.639,154.808
C03464=1061.668,-109.086,438.799,171.359,25.639,154.808
C03465=1061.661,-109.336,438.808,171.357,25.637,154.808
C03466=1061.655,-109.585,438.819,171.355,25.637,154.808
C03467=1061.649,-109.835,438.828,171.353,25.636,154.808
C03468=1061.643,-110.085,438.838,171.352,25.634,154.808
C03469=1061.636,-110.334,438.847,171.350,25.634,154.808
C03470=1061.630,-110.584,438.857,171.348,25.633,154.808
C03471=1061.625,-110.834,438.867,171.346,25.632,154.808
C03472=1061.618,-111.084,438.877,171.345,25.631,154.808
C03473=1061.612,-111.333,438.887,171.343,25.630,154.808
C03474=1061.606,-111.583,438.896,171.341,25.629,154.808
C03475=1061.600,-111.833,438.906,171.339,25.628,154.808
C03476=1061.594,-112.083,438.916,171.337,25.627,154.808
C03477=1061.587,-112.333,438.925,171.336,25.626,154.808
C03478=1061.581,-112.582,438.935,171.334,25.625,154.809
C03479=1061.575,-112.831,438.945,171.332,25.624,154.809
C03480=1061.569,-113.081,438.955,171.330,25.624,154.809
C03481=1061.562,-113.331,438.964,171.328,25.622,154.809
C03482=1061.556,-113.581,438.974,171.326,25.622,154.809
C03483=1061.551,-113.831,438.984,171.324,25.620,154.809
C03484=1061.545,-114.081,438.993,171.322,25.620,154.809
C03485=1061.537,-114.363,439.004,171.320,25.619,154.809
C03486=1061.531,-114.646,439.015,171.319,25.618,154.809
C03487=1061.523,-114.928,439.026,171.316,25.616,154.809
C03488=1061.517,-115.211,439.036,171.314,25.616,154.809
C03489=1061.511,-115.461,439.046,171.312,25.615,154.809
C03490=1061.505,-115.711,439.056,171.310,25.614,154.809
C03491=1061.498,-115.961,439.065,171.309,25.613,154.809
C03492=1061.492,-116.210,439.075,171.307,25.612,154.809
C03493=1061.487,-116.460,439.084,171.305,25.612,154.809
C03494=1061.481,-116.709,439.093,171.303,25.610,154.809
C03495=1061.474,-116.959,439.103,171.301,25.610,154.809
C03496=1061.468,-117.209,439.113,171.300,25.609,154.810
C03497=1061.461,-117.458,439.122,171.298,25.608,154.810
C03498=1061.455,-117.708,439.131,171.296,25.607,154.810
C03499=1061.449,-117.958,439.141,171.294,25.607,154.810
C03500=1061.443,-118.208,439.150,171.292,25.606,154.810
C03501=1061.437,-118.458,439.160,171.290,25.605,154.810
C03502=1061.430,-118.707,439.169,171.288,25.604,154.810
C03503=1061.424,-118.957,439.179,171.286,25.603,154.810
C03504=1061.419,-119.206,439.188,171.284,25.602,154.810
C03505=1061.412,-119.456,439.198,171.282,25.602,154.810
C03506=1061.406,-119.706,439.207,171.281,25.600,154.810
C03507=1061.400,-119.956,439.216,171.279,25.600,154.810
C03508=1061.394,-120.206,439.226,171.277,25.599,154.810
C03509=1061.387,-120.456,439.235,171.275,25.599,154.810
C03510=1061.381,-120.705,439.244,171.273,25.597,154.810
C03511=1061.375,-120.955,439.254,171.271,25.597,154.811
C03512=1061.369,-121.204,439.263,171.270,25.596,154.811
C03513=1061.363,-121.454,439.273,171.268,25.596,154.811
C03514=1061.357,-121.704,439.282,171.266,25.594,154.811
C03515=1061.351,-121.954,439.291,171.264,25.594,154.811
C03516=1061.344,-122.204,439.300,171.262,25.593,154.811
C03517=1061.338,-122.454,439.310,171.260,25.593,154.811
C03518=1061.332,-122.703,439.319,171.258,25.592,154.811
C03519=1061.326,-122.952,439.328,171.257,25.591,154.811
C03520=1061.321,-123.203,439.337,171.255,25.590,154.811
C03521=1061.314,-123.453,439.347,171.253,25.590,154.811
C03522=1061.308,-123.702,439.356,171.251,25.589,154.811
C03523=1061.301,-123.952,439.365,171.249,25.588,154.812
C03524=1061.296,-124.201,439.374,171.247,25.588,154.812
C03525=1061.290,-124.451,439.383,171.246,25.587,154.812
C03526=1061.284,-124.701,439.393,171.244,25.586,154.812
C03527=1061.277,-124.951,439.402,171.242,25.585,154.812
C03528=1061.271,-125.201,439.411,171.240,25.585,154.812
C03529=1061.265,-125.451,439.420,171.237,25.584,154.812
C03530=1061.259,-125.700,439.429,171.236,25.583,154.812
C03531=1061.252,-125.950,439.438,171.234,25.583,154.812
C03532=1061.246,-126.200,439.447,171.232,25.582,154.812
C03533=1061.240,-126.450,439.457,171.230,25.581,154.813
C03534=1061.234,-126.700,439.466,171.228,25.581,154.813
C03535=1061.228,-126.948,439.475,171.226,25.580,154.813
C03536=1061.222,-127.199,439.484,171.224,25.580,154.813
C03537=1061.216,-127.449,439.493,171.223,25.579,154.813
C03538=1061.209,-127.698,439.502,171.221,25.578,154.813
C03539=1061.204,-127.948,439.511,171.219,25.577,154.813
C03540=1061.199,-128.198,439.522,171.217,25.576,154.813
C03541=1061.196,-128.449,439.532,171.216,25.574,154.813
C03542=1061.195,-128.699,439.543,171.214,25.572,154.813
C03543=1061.194,-128.950,439.555,171.214,25.569,154.812
C03544=1061.196,-129.200,439.569,171.213,25.565,154.812
C03545=1061.199,-129.453,439.582,171.212,25.560,154.811
C03546=1061.203,-129.703,439.597,171.211,25.555,154.810
C03547=1061.209,-129.954,439.611,171.211,25.550,154.809
C03548=1061.216,-130.205,439.627,171.210,25.544,154.808
C03549=1060.836,-130.227,439.436,171.163,25.701,154.841
C03550=1060.829,-129.977,439.420,171.163,25.707,154.842
C03551=1060.823,-129.726,439.405,171.163,25.712,154.843
C03552=1060.819,-129.475,439.390,171.164,25.717,154.844
C03553=1060.816,-129.223,439.377,171.165,25.722,154.845
C03554=1060.815,-128.973,439.364,171.165,25.725,154.845
C03555=1060.814,-128.722,439.352,171.167,25.728,154.846
C03556=1060.816,-128.471,439.340,171.168,25.731,154.846
C03557=1060.819,-128.221,439.329,171.170,25.733,154.846
C03558=1060.823,-127.970,439.320,171.171,25.734,154.846
C03559=1060.829,-127.721,439.310,171.173,25.735,154.846
C03560=1060.835,-127.472,439.301,171.175,25.735,154.846
C03561=1060.841,-127.221,439.293,171.177,25.736,154.846
C03562=1060.847,-126.972,439.283,171.179,25.737,154.846
C03563=1060.854,-126.722,439.273,171.181,25.737,154.846
C03564=1060.859,-126.473,439.264,171.182,25.738,154.846
C03565=1060.866,-126.223,439.256,171.184,25.738,154.846
C03566=1060.872,-125.973,439.246,171.186,25.739,154.845
C03567=1060.878,-125.723,439.237,171.188,25.740,154.845
C03568=1060.885,-125.473,439.229,171.190,25.740,154.845
C03569=1060.890,-125.224,439.219,171.192,25.741,154.845
C03570=1060.896,-124.974,439.210,171.194,25.742,154.845
C03571=1060.903,-124.724,439.200,171.196,25.743,154.845
C03572=1060.909,-124.474,439.192,171.198,25.744,154.845
C03573=1060.915,-124.224,439.182,171.200,25.744,154.845
C03574=1060.922,-123.975,439.173,171.202,25.745,154.845
C03575=1060.927,-123.725,439.164,171.204,25.745,154.845
C03576=1060.933,-123.475,439.155,171.206,25.746,154.844
C03577=1060.940,-123.226,439.146,171.207,25.747,154.844
C03578=1060.946,-122.976,439.136,171.209,25.748,154.844
C03579=1060.952,-122.726,439.127,171.211,25.748,154.844
C03580=1060.958,-122.476,439.117,171.213,25.749,154.844
C03581=1060.964,-122.226,439.109,171.215,25.750,154.844
C03582=1060.970,-121.977,439.099,171.217,25.750,154.844
C03583=1060.976,-121.727,439.090,171.218,25.751,154.844
C03584=1060.983,-121.477,439.081,171.220,25.752,154.844
C03585=1060.989,-121.228,439.071,171.222,25.753,154.844
C03586=1060.995,-120.978,439.061,171.224,25.753,154.844
C03587=1061.001,-120.728,439.053,171.226,25.754,154.844
C03588=1061.007,-120.478,439.043,171.228,25.755,154.844
C03589=1061.013,-120.228,439.034,171.229,25.756,154.843
C03590=1061.019,-119.979,439.024,171.231,25.756,154.843
C03591=1061.025,-119.729,439.015,171.233,25.757,154.843
C03592=1061.031,-119.479,439.005,171.235,25.758,154.843
C03593=1061.038,-119.230,438.996,171.238,25.759,154.843
C03594=1061.045,-118.980,438.987,171.240,25.759,154.843
C03595=1061.051,-118.730,438.977,171.241,25.761,154.843
C03596=1061.056,-118.481,438.968,171.243,25.761,154.843
C03597=1061.062,-118.231,438.958,171.245,25.762,154.843
C03598=1061.068,-117.981,438.949,171.247,25.763,154.843
C03599=1061.074,-117.731,438.940,171.249,25.764,154.843
C03600=1061.081,-117.481,438.930,171.250,25.764,154.843
C03601=1061.087,-117.231,438.921,171.252,25.765,154.843
C03602=1061.093,-116.981,438.911,171.254,25.766,154.843
C03603=1061.099,-116.732,438.902,171.256,25.767,154.842
C03604=1061.105,-116.482,438.892,171.258,25.768,154.842
C03605=1061.112,-116.232,438.882,171.259,25.768,154.842
C03606=1061.118,-115.982,438.873,171.261,25.770,154.842
C03607=1061.124,-115.732,438.863,171.263,25.770,154.842
C03608=1061.129,-115.483,438.854,171.265,25.771,154.842
C03609=1061.136,-115.234,438.844,171.267,25.772,154.842
C03610=1061.144,-114.951,438.833,171.269,25.773,154.842
C03611=1061.150,-114.668,438.823,171.271,25.774,154.842
C03612=1061.158,-114.385,438.812,171.273,25.775,154.842
C03613=1061.164,-114.102,438.801,171.276,25.776,154.842
C03614=1061.170,-113.853,438.791,171.278,25.777,154.842
C03615=1061.177,-113.603,438.781,171.279,25.778,154.842
C03616=1061.183,-113.354,438.772,171.281,25.779,154.842
C03617=1061.189,-113.104,438.762,171.283,25.780,154.842
C03618=1061.195,-112.854,438.753,171.285,25.780,154.842
C03619=1061.201,-112.604,438.743,171.286,25.781,154.842
C03620=1061.207,-112.354,438.733,171.288,25.782,154.842
C03621=1061.214,-112.105,438.724,171.290,25.783,154.842
C03622=1061.219,-111.855,438.714,171.292,25.784,154.841
C03623=1061.225,-111.605,438.704,171.294,25.785,154.842
C03624=1061.232,-111.356,438.694,171.296,25.786,154.841
C03625=1061.237,-111.107,438.685,171.297,25.787,154.841
C03626=1061.243,-110.857,438.675,171.299,25.788,154.841
C03627=1061.250,-110.606,438.665,171.301,25.789,154.841
C03628=1061.256,-110.356,438.656,171.303,25.790,154.841
C03629=1061.263,-110.107,438.646,171.304,25.790,154.841
C03630=1061.268,-109.892,438.637,171.306,25.792,154.841
C03631=1061.273,-109.677,438.629,171.308,25.792,154.841
C03632=1061.279,-109.462,438.620,171.310,25.793,154.841
